SPLINE
SPL {X  -156.487, Y  +349.204, Z    +0.000, E1   +21.338, E3 +377036.669}
SPL {X  -159.136, Y  +365.992, Z    +0.000, E1   +12.463, E3 +377047.428}
SPL {X  -159.799, Y  +374.694, Z    +0.000, E1    +7.504, E3 +377050.531}
SPL {X  -159.976, Y  +380.404, Z    +0.000, E1    +3.959, E3 +377052.064}
SPL {X  -159.990, Y  +384.773, Z    +0.000, E1    +1.003, E3 +377052.959}
SPL {X  -159.990, Y  +387.968, Z    +0.000, E1    -1.448, E3 +377053.527}
SPL {X  -159.990, Y  +391.397, Z    +0.000, E1    -4.422, E3 +377054.151}
SPL {X  -159.990, Y  +395.864, Z    +0.000, E1    -8.712, E3 +377055.240}
SPL {X  -159.990, Y  +401.273, Z    +0.000, E1   -14.176, E3 +377056.967}
SPL {X  -159.990, Y  +409.369, Z    +0.000, E1   -21.807, E3 +377060.759}
SPL {X  -159.990, Y  +436.107, Z    +0.000, E1   -36.921, E3 +377083.684}
SPL {X  -159.990, Y  +469.969, Z    +0.000, E1   -41.961, E3 +377138.388}
SPL {X  -159.990, Y  +477.498, Z    +0.000, E1   -41.916, E3 +377156.272}
SPL {X  -159.990, Y  +483.140, Z    +0.000, E1   -41.902, E3 +377169.628}
SPL {X  -159.990, Y  +488.618, Z    +0.000, E1   -41.913, E3 +377182.559}
SPL {X  -159.990, Y  +494.299, Z    +0.000, E1   -41.910, E3 +377195.994}
SPL {X  -159.990, Y  +499.538, Z    +0.000, E1   -41.904, E3 +377208.388}
SPL {X  -159.990, Y  +505.259, Z    +0.000, E1   -41.922, E3 +377221.887}
SPL {X  -159.990, Y  +511.862, Z    +0.000, E1   -41.927, E3 +377237.498}
SPL {X  -159.990, Y  +519.146, Z    +0.000, E1   -41.942, E3 +377254.691}
SPL {X  -159.990, Y  +526.974, Z    +0.000, E1   -41.950, E3 +377273.191}
SPL {X  -159.990, Y  +533.758, Z    +0.000, E1   -41.910, E3 +377289.294}
SPL {X  -159.990, Y  +539.474, Z    +0.000, E1   -41.912, E3 +377302.821}
SPL {X  -159.990, Y  +544.879, Z    +0.000, E1   -41.899, E3 +377315.633}
SPL {X  -159.990, Y  +550.802, Z    +0.000, E1   -41.920, E3 +377329.614}
SPL {X  -159.990, Y  +556.952, Z    +0.000, E1   -41.911, E3 +377344.153}
SPL {X  -159.990, Y  +562.629, Z    +0.000, E1   -41.910, E3 +377357.571}
SPL {X  -159.990, Y  +567.682, Z    +0.000, E1   -41.901, E3 +377369.530}
SPL {X  -159.990, Y  +572.912, Z    +0.000, E1   -41.914, E3 +377381.877}
SPL {X  -159.990, Y  +578.863, Z    +0.000, E1   -41.918, E3 +377395.941}
SPL {X  -159.990, Y  +584.320, Z    +0.000, E1   -41.901, E3 +377408.888}
SPL {X  -159.990, Y  +589.217, Z    +0.000, E1   -41.901, E3 +377420.461}
SPL {X  -159.990, Y  +594.252, Z    +0.000, E1   -41.903, E3 +377432.376}
SPL {X  -159.990, Y  +600.237, Z    +0.000, E1   -41.928, E3 +377446.493}
SPL {X  -159.990, Y  +607.478, Z    +0.000, E1   -41.933, E3 +377463.602}
SPL {X  -159.990, Y  +614.570, Z    +0.000, E1   -41.926, E3 +377480.383}
SPL {X  -159.990, Y  +621.417, Z    +0.000, E1   -41.931, E3 +377496.576}
SPL {X  -159.990, Y  +627.900, Z    +0.000, E1   -41.914, E3 +377511.916}
SPL {X  -159.990, Y  +634.411, Z    +0.000, E1   -41.931, E3 +377527.285}
SPL {X  -159.990, Y  +641.479, Z    +0.000, E1   -41.931, E3 +377544.002}
SPL {X  -159.990, Y  +647.782, Z    +0.000, E1   -41.914, E3 +377558.923}
SPL {X  -159.990, Y  +653.094, Z    +0.000, E1   -41.905, E3 +377571.502}
SPL {X  -159.990, Y  +657.893, Z    +0.000, E1   -41.899, E3 +377582.867}
SPL {X  -159.990, Y  +662.516, Z    +0.000, E1   -41.899, E3 +377593.799}
SPL {X  -159.990, Y  +668.411, Z    +0.000, E1   -41.929, E3 +377607.692}
SPL {X  -159.968, Y  +674.139, Z    +0.000, E1   -41.898, E3 +377621.296}
SPL {X  -159.817, Y  +678.937, Z    +0.000, E1   -41.879, E3 +377632.793}
SPL {X  -159.484, Y  +684.213, Z    +0.000, E1   -41.818, E3 +377645.629}
SPL {X  -159.007, Y  +689.209, Z    +0.000, E1   -41.732, E3 +377657.934}
SPL {X  -158.327, Y  +694.511, Z    +0.000, E1   -41.622, E3 +377671.184}
SPL {X  -157.480, Y  +699.729, Z    +0.000, E1   -41.453, E3 +377684.447}
SPL {X  -156.604, Y  +704.242, Z    +0.000, E1   -41.288, E3 +377696.056}
SPL {X  -155.514, Y  +709.078, Z    +0.000, E1   -41.107, E3 +377708.610}
SPL {X  -154.232, Y  +714.035, Z    +0.000, E1   -40.861, E3 +377721.669}
SPL {X  -153.147, Y  +717.790, Z    +0.000, E1   -40.640, E3 +377731.687}
SPL {X  -151.881, Y  +721.788, Z    +0.000, E1   -40.435, E3 +377742.374}
SPL {X  -148.572, Y  +730.857, Z    +0.000, E1   -36.304, E3 +377798.582}
ENDSPLINE

SPLINE
SPL {X  -156.377, Y  +705.307, Z    +0.000, E1   -21.740, E3 +377852.831}
SPL {X  -159.301, Y  +686.331, Z    +0.000, E1   -11.648, E3 +377865.476}
SPL {X  -159.936, Y  +675.651, Z    +0.000, E1    -5.377, E3 +377869.192}
SPL {X  -159.990, Y  +670.142, Z    +0.000, E1    -1.740, E3 +377870.491}
SPL {X  -159.990, Y  +666.629, Z    +0.000, E1    +0.827, E3 +377871.140}
SPL {X  -159.990, Y  +662.407, Z    +0.000, E1    +4.406, E3 +377871.991}
SPL {X  -159.990, Y  +655.884, Z    +0.000, E1   +10.601, E3 +377873.856}
SPL {X  -159.990, Y  +646.242, Z    +0.000, E1   +19.956, E3 +377877.775}
SPL {X  -159.990, Y  +624.365, Z    +0.000, E1   +33.860, E3 +377895.677}
SPL {X  -159.990, Y  +615.596, Z    +0.000, E1   +36.980, E3 +377905.336}
SPL {X  -159.990, Y  +586.905, Z    +0.000, E1   +41.264, E3 +377952.362}
SPL {X  -159.990, Y  +581.111, Z    +0.000, E1   +41.245, E3 +377966.416}
SPL {X  -159.990, Y  +576.269, Z    +0.000, E1   +41.239, E3 +377978.143}
SPL {X  -159.990, Y  +571.714, Z    +0.000, E1   +41.240, E3 +377989.171}
SPL {X  -159.990, Y  +567.050, Z    +0.000, E1   +41.238, E3 +378000.458}
SPL {X  -159.990, Y  +561.959, Z    +0.000, E1   +41.251, E3 +378012.757}
SPL {X  -159.990, Y  +557.719, Z    +0.000, E1   +41.226, E3 +378023.059}
SPL {X  -159.990, Y  +554.148, Z    +0.000, E1   +41.237, E3 +378031.674}
SPL {X  -159.990, Y  +548.812, Z    +0.000, E1   +41.263, E3 +378044.549}
SPL {X  -159.990, Y  +542.097, Z    +0.000, E1   +41.274, E3 +378060.801}
SPL {X  -159.990, Y  +535.325, Z    +0.000, E1   +41.260, E3 +378077.202}
SPL {X  -159.990, Y  +529.136, Z    +0.000, E1   +41.262, E3 +378092.170}
SPL {X  -159.990, Y  +524.776, Z    +0.000, E1   +41.225, E3 +378102.783}
SPL {X  -159.990, Y  +521.454, Z    +0.000, E1   +41.236, E3 +378110.805}
SPL {X  -159.990, Y  +515.605, Z    +0.000, E1   +41.288, E3 +378124.844}
SPL {X  -159.990, Y  +509.898, Z    +0.000, E1   +41.246, E3 +378138.706}
SPL {X  -159.990, Y  +505.215, Z    +0.000, E1   +41.261, E3 +378150.022}
SPL {X  -159.990, Y  +500.102, Z    +0.000, E1   +41.251, E3 +378162.405}
SPL {X  -159.990, Y  +495.023, Z    +0.000, E1   +41.263, E3 +378174.654}
SPL {X  -159.990, Y  +479.011, Z    +0.000, E1   +45.740, E3 +378184.036}
SPL {X  -159.990, Y  +471.379, Z    +0.000, E1   +46.435, E3 +378195.651}
SPL {X  -159.990, Y  +466.895, Z    +0.000, E1   +45.533, E3 +378210.056}
SPL {X  -159.990, Y  +462.409, Z    +0.000, E1   +44.664, E3 +378224.831}
SPL {X  -159.990, Y  +458.229, Z    +0.000, E1   +43.579, E3 +378240.313}
SPL {X  -159.990, Y  +453.434, Z    +0.000, E1   +43.227, E3 +378253.087}
SPL {X  -159.990, Y  +448.702, Z    +0.000, E1   +43.218, E3 +378263.809}
SPL {X  -159.990, Y  +442.224, Z    +0.000, E1   +43.270, E3 +378278.359}
SPL {X  -159.990, Y  +435.724, Z    +0.000, E1   +43.218, E3 +378293.117}
SPL {X  -159.990, Y  +430.527, Z    +0.000, E1   +43.236, E3 +378304.807}
SPL {X  -159.990, Y  +424.433, Z    +0.000, E1   +43.237, E3 +378318.556}
SPL {X  -159.990, Y  +419.466, Z    +0.000, E1   +43.217, E3 +378329.795}
SPL {X  -159.990, Y  +414.585, Z    +0.000, E1   +43.233, E3 +378340.787}
SPL {X  -159.990, Y  +409.927, Z    +0.000, E1   +43.217, E3 +378351.319}
SPL {X  -159.990, Y  +405.428, Z    +0.000, E1   +43.230, E3 +378361.477}
SPL {X  -159.990, Y  +398.518, Z    +0.000, E1   +43.261, E3 +378377.032}
SPL {X  -159.990, Y  +392.163, Z    +0.000, E1   +43.223, E3 +378391.432}
SPL {X  -159.990, Y  +387.342, Z    +0.000, E1   +43.224, E3 +378402.309}
SPL {X  -159.990, Y  +382.548, Z    +0.000, E1   +43.224, E3 +378413.132}
SPL {X  -159.922, Y  +377.835, Z    +0.000, E1   +43.211, E3 +378423.849}
SPL {X  -159.608, Y  +371.448, Z    +0.000, E1   +43.200, E3 +378438.525}
SPL {X  -158.905, Y  +363.898, Z    +0.000, E1   +43.073, E3 +378456.293}
SPL {X  -158.182, Y  +358.518, Z    +0.000, E1   +42.902, E3 +378469.237}
SPL {X  -157.507, Y  +354.423, Z    +0.000, E1   +42.786, E3 +378479.182}
SPL {X  -156.676, Y  +350.104, Z    +0.000, E1   +42.637, E3 +378489.787}
SPL {X  -155.489, Y  +344.819, Z    +0.000, E1   +42.446, E3 +378502.911}
SPL {X  -153.911, Y  +338.816, Z    +0.000, E1   +42.155, E3 +378518.087}
SPL {X  -152.412, Y  +333.846, Z    +0.000, E1   +41.856, E3 +378530.857}
SPL {X  -151.009, Y  +329.651, Z    +0.000, E1   +41.581, E3 +378541.757}
SPL {X  -148.356, Y  +322.607, Z    +0.000, E1   +36.121, E3 +378602.233}
ENDSPLINE

SPLINE
SPL {X  -156.487, Y  +349.204, Z    +0.000, E1   +21.338, E3 +378657.359}
SPL {X  -159.136, Y  +365.992, Z    +0.000, E1   +12.463, E3 +378668.117}
SPL {X  -159.799, Y  +374.694, Z    +0.000, E1    +7.504, E3 +378671.221}
SPL {X  -159.976, Y  +380.404, Z    +0.000, E1    +3.959, E3 +378672.754}
SPL {X  -159.990, Y  +384.773, Z    +0.000, E1    +1.003, E3 +378673.648}
SPL {X  -159.990, Y  +387.968, Z    +0.000, E1    -1.448, E3 +378674.217}
SPL {X  -159.990, Y  +391.397, Z    +0.000, E1    -4.422, E3 +378674.841}
SPL {X  -159.990, Y  +395.864, Z    +0.000, E1    -8.712, E3 +378675.929}
SPL {X  -159.990, Y  +401.273, Z    +0.000, E1   -14.176, E3 +378677.657}
SPL {X  -159.990, Y  +409.369, Z    +0.000, E1   -21.807, E3 +378681.448}
SPL {X  -159.990, Y  +436.107, Z    +0.000, E1   -36.921, E3 +378704.374}
SPL {X  -159.990, Y  +469.969, Z    +0.000, E1   -41.961, E3 +378759.078}
SPL {X  -159.990, Y  +477.498, Z    +0.000, E1   -41.916, E3 +378776.962}
SPL {X  -159.990, Y  +483.140, Z    +0.000, E1   -41.902, E3 +378790.317}
SPL {X  -159.990, Y  +488.618, Z    +0.000, E1   -41.913, E3 +378803.249}
SPL {X  -159.990, Y  +494.299, Z    +0.000, E1   -41.910, E3 +378816.683}
SPL {X  -159.990, Y  +499.538, Z    +0.000, E1   -41.904, E3 +378829.078}
SPL {X  -159.990, Y  +504.097, Z    +0.000, E1   -41.897, E3 +378839.866}
SPL {X  -159.990, Y  +509.413, Z    +0.000, E1   -41.921, E3 +378852.401}
SPL {X  -159.990, Y  +516.193, Z    +0.000, E1   -41.932, E3 +378868.417}
SPL {X  -159.990, Y  +523.027, Z    +0.000, E1   -41.926, E3 +378884.579}
SPL {X  -159.990, Y  +528.611, Z    +0.000, E1   -41.900, E3 +378897.834}
SPL {X  -159.990, Y  +533.758, Z    +0.000, E1   -41.910, E3 +378909.983}
SPL {X  -159.990, Y  +539.474, Z    +0.000, E1   -41.912, E3 +378923.511}
SPL {X  -159.990, Y  +544.879, Z    +0.000, E1   -41.899, E3 +378936.322}
SPL {X  -159.990, Y  +550.802, Z    +0.000, E1   -41.920, E3 +378950.304}
SPL {X  -159.990, Y  +556.952, Z    +0.000, E1   -41.911, E3 +378964.843}
SPL {X  -159.990, Y  +562.629, Z    +0.000, E1   -41.910, E3 +378978.261}
SPL {X  -159.990, Y  +567.682, Z    +0.000, E1   -41.901, E3 +378990.220}
SPL {X  -159.990, Y  +574.350, Z    +0.000, E1   -41.955, E3 +379005.905}
SPL {X  -159.990, Y  +580.118, Z    +0.000, E1   -41.891, E3 +379019.642}
SPL {X  -159.990, Y  +584.320, Z    +0.000, E1   -41.901, E3 +379029.578}
SPL {X  -159.990, Y  +589.217, Z    +0.000, E1   -41.901, E3 +379041.151}
SPL {X  -159.990, Y  +594.252, Z    +0.000, E1   -41.903, E3 +379053.065}
SPL {X  -159.990, Y  +600.237, Z    +0.000, E1   -41.928, E3 +379067.183}
SPL {X  -159.990, Y  +605.518, Z    +0.000, E1   -41.890, E3 +379079.721}
SPL {X  -159.990, Y  +610.545, Z    +0.000, E1   -41.917, E3 +379091.569}
SPL {X  -159.990, Y  +615.720, Z    +0.000, E1   -41.899, E3 +379103.829}
SPL {X  -159.990, Y  +620.005, Z    +0.000, E1   -41.900, E3 +379113.962}
SPL {X  -159.990, Y  +624.919, Z    +0.000, E1   -41.912, E3 +379125.569}
SPL {X  -159.990, Y  +629.282, Z    +0.000, E1   -41.888, E3 +379135.910}
SPL {X  -159.990, Y  +632.270, Z    +0.000, E1   -41.887, E3 +379142.982}
SPL {X  -159.990, Y  +637.009, Z    +0.000, E1   -41.925, E3 +379154.124}
SPL {X  -159.990, Y  +642.624, Z    +0.000, E1   -41.901, E3 +379167.445}
SPL {X  -159.990, Y  +647.782, Z    +0.000, E1   -41.914, E3 +379179.613}
SPL {X  -159.990, Y  +653.094, Z    +0.000, E1   -41.905, E3 +379192.191}
SPL {X  -159.990, Y  +657.893, Z    +0.000, E1   -41.899, E3 +379203.557}
SPL {X  -159.990, Y  +662.516, Z    +0.000, E1   -41.899, E3 +379214.488}
SPL {X  -159.990, Y  +666.974, Z    +0.000, E1   -41.897, E3 +379225.033}
SPL {X  -159.984, Y  +672.859, Z    +0.000, E1   -41.934, E3 +379238.894}
SPL {X  -159.817, Y  +678.937, Z    +0.000, E1   -41.879, E3 +379253.482}
SPL {X  -159.484, Y  +684.213, Z    +0.000, E1   -41.818, E3 +379266.318}
SPL {X  -159.007, Y  +689.209, Z    +0.000, E1   -41.732, E3 +379278.623}
SPL {X  -158.485, Y  +693.390, Z    +0.000, E1   -41.627, E3 +379289.076}
SPL {X  -157.663, Y  +698.690, Z    +0.000, E1   -41.523, E3 +379302.438}
SPL {X  -156.604, Y  +704.242, Z    +0.000, E1   -41.288, E3 +379316.746}
SPL {X  -155.831, Y  +707.744, Z    +0.000, E1   -41.132, E3 +379325.866}
SPL {X  -155.167, Y  +710.488, Z    +0.000, E1   -41.008, E3 +379333.044}
SPL {X  -154.232, Y  +714.035, Z    +0.000, E1   -40.861, E3 +379342.358}
SPL {X  -153.147, Y  +717.790, Z    +0.000, E1   -40.640, E3 +379352.377}
SPL {X  -151.881, Y  +721.788, Z    +0.000, E1   -40.435, E3 +379363.063}
SPL {X  -148.572, Y  +730.857, Z    +0.000, E1   -36.304, E3 +379419.272}
ENDSPLINE

SPLINE
SPL {X  -156.377, Y  +705.307, Z    +0.000, E1   -21.740, E3 +379473.521}
SPL {X  -158.965, Y  +689.585, Z    +0.000, E1   -13.405, E3 +379484.678}
SPL {X  -159.884, Y  +677.314, Z    +0.000, E1    -6.475, E3 +379489.391}
SPL {X  -159.990, Y  +670.142, Z    +0.000, E1    -1.740, E3 +379491.180}
SPL {X  -159.990, Y  +666.629, Z    +0.000, E1    +0.827, E3 +379491.830}
SPL {X  -159.990, Y  +662.407, Z    +0.000, E1    +4.406, E3 +379492.680}
SPL {X  -159.990, Y  +655.884, Z    +0.000, E1   +10.601, E3 +379494.546}
SPL {X  -159.990, Y  +643.833, Z    +0.000, E1   +21.883, E3 +379500.175}
SPL {X  -159.990, Y  +617.235, Z    +0.000, E1   +36.481, E3 +379524.075}
SPL {X  -159.990, Y  +586.905, Z    +0.000, E1   +41.264, E3 +379573.051}
SPL {X  -159.990, Y  +581.111, Z    +0.000, E1   +41.245, E3 +379587.105}
SPL {X  -159.990, Y  +576.269, Z    +0.000, E1   +41.239, E3 +379598.833}
SPL {X  -159.990, Y  +571.714, Z    +0.000, E1   +41.240, E3 +379609.861}
SPL {X  -159.990, Y  +567.050, Z    +0.000, E1   +41.238, E3 +379621.148}
SPL {X  -159.990, Y  +561.959, Z    +0.000, E1   +41.251, E3 +379633.446}
SPL {X  -159.990, Y  +557.719, Z    +0.000, E1   +41.226, E3 +379643.749}
SPL {X  -159.990, Y  +554.148, Z    +0.000, E1   +41.237, E3 +379652.364}
SPL {X  -159.990, Y  +548.812, Z    +0.000, E1   +41.263, E3 +379665.238}
SPL {X  -159.990, Y  +543.804, Z    +0.000, E1   +41.237, E3 +379677.403}
SPL {X  -159.990, Y  +538.952, Z    +0.000, E1   +41.247, E3 +379689.150}
SPL {X  -159.990, Y  +534.225, Z    +0.000, E1   +41.236, E3 +379700.584}
SPL {X  -159.990, Y  +529.136, Z    +0.000, E1   +41.262, E3 +379712.859}
SPL {X  -159.990, Y  +522.690, Z    +0.000, E1   +41.265, E3 +379728.459}
SPL {X  -159.990, Y  +516.698, Z    +0.000, E1   +41.259, E3 +379742.933}
SPL {X  -159.990, Y  +510.896, Z    +0.000, E1   +41.267, E3 +379756.951}
SPL {X  -159.990, Y  +505.215, Z    +0.000, E1   +41.261, E3 +379770.711}
SPL {X  -159.990, Y  +500.102, Z    +0.000, E1   +41.251, E3 +379783.094}
SPL {X  -159.990, Y  +495.023, Z    +0.000, E1   +41.263, E3 +379795.343}
SPL {X  -159.990, Y  +479.011, Z    +0.000, E1   +45.740, E3 +379804.725}
SPL {X  -159.990, Y  +471.379, Z    +0.000, E1   +46.435, E3 +379816.341}
SPL {X  -159.990, Y  +466.895, Z    +0.000, E1   +45.533, E3 +379830.745}
SPL {X  -159.990, Y  +462.409, Z    +0.000, E1   +44.664, E3 +379845.520}
SPL {X  -159.990, Y  +458.229, Z    +0.000, E1   +43.579, E3 +379861.003}
SPL {X  -159.990, Y  +453.434, Z    +0.000, E1   +43.227, E3 +379873.777}
SPL {X  -159.990, Y  +448.702, Z    +0.000, E1   +43.218, E3 +379884.499}
SPL {X  -159.990, Y  +444.476, Z    +0.000, E1   +43.219, E3 +379894.037}
SPL {X  -159.990, Y  +440.246, Z    +0.000, E1   +43.217, E3 +379903.595}
SPL {X  -159.990, Y  +434.411, Z    +0.000, E1   +43.246, E3 +379916.725}
SPL {X  -159.990, Y  +429.216, Z    +0.000, E1   +43.210, E3 +379928.498}
SPL {X  -159.990, Y  +424.433, Z    +0.000, E1   +43.237, E3 +379939.245}
SPL {X  -159.990, Y  +419.466, Z    +0.000, E1   +43.217, E3 +379950.485}
SPL {X  -159.990, Y  +414.585, Z    +0.000, E1   +43.233, E3 +379961.477}
SPL {X  -159.990, Y  +409.927, Z    +0.000, E1   +43.217, E3 +379972.009}
SPL {X  -159.990, Y  +405.428, Z    +0.000, E1   +43.230, E3 +379982.167}
SPL {X  -159.990, Y  +398.518, Z    +0.000, E1   +43.261, E3 +379997.721}
SPL {X  -159.990, Y  +392.163, Z    +0.000, E1   +43.223, E3 +380012.121}
SPL {X  -159.990, Y  +387.342, Z    +0.000, E1   +43.224, E3 +380022.999}
SPL {X  -159.990, Y  +382.548, Z    +0.000, E1   +43.224, E3 +380033.821}
SPL {X  -159.922, Y  +377.835, Z    +0.000, E1   +43.211, E3 +380044.538}
SPL {X  -159.712, Y  +373.072, Z    +0.000, E1   +43.177, E3 +380055.504}
SPL {X  -159.289, Y  +367.537, Z    +0.000, E1   +43.118, E3 +380068.416}
SPL {X  -158.730, Y  +362.464, Z    +0.000, E1   +43.003, E3 +380080.448}
SPL {X  -158.182, Y  +358.518, Z    +0.000, E1   +42.902, E3 +380089.926}
SPL {X  -157.507, Y  +354.423, Z    +0.000, E1   +42.786, E3 +380099.872}
SPL {X  -156.676, Y  +350.104, Z    +0.000, E1   +42.637, E3 +380110.477}
SPL {X  -155.807, Y  +346.154, Z    +0.000, E1   +42.470, E3 +380120.304}
SPL {X  -154.777, Y  +341.993, Z    +0.000, E1   +42.302, E3 +380130.729}
SPL {X  -153.585, Y  +337.686, Z    +0.000, E1   +42.062, E3 +380141.705}
SPL {X  -152.412, Y  +333.846, Z    +0.000, E1   +41.856, E3 +380151.547}
SPL {X  -151.009, Y  +329.651, Z    +0.000, E1   +41.581, E3 +380162.447}
SPL {X  -148.356, Y  +322.607, Z    +0.000, E1   +36.121, E3 +380222.923}
ENDSPLINE

SPLINE
SPL {X  -156.487, Y  +349.204, Z    +0.000, E1   +21.338, E3 +380278.048}
SPL {X  -159.136, Y  +365.992, Z    +0.000, E1   +12.463, E3 +380288.807}
SPL {X  -159.799, Y  +374.694, Z    +0.000, E1    +7.504, E3 +380291.911}
SPL {X  -159.976, Y  +380.404, Z    +0.000, E1    +3.959, E3 +380293.444}
SPL {X  -159.990, Y  +384.773, Z    +0.000, E1    +1.003, E3 +380294.338}
SPL {X  -159.990, Y  +387.968, Z    +0.000, E1    -1.448, E3 +380294.906}
SPL {X  -159.990, Y  +391.397, Z    +0.000, E1    -4.422, E3 +380295.530}
SPL {X  -159.990, Y  +395.864, Z    +0.000, E1    -8.712, E3 +380296.619}
SPL {X  -159.990, Y  +401.273, Z    +0.000, E1   -14.176, E3 +380298.346}
SPL {X  -159.990, Y  +411.788, Z    +0.000, E1   -23.693, E3 +380303.889}
SPL {X  -159.990, Y  +438.158, Z    +0.000, E1   -37.630, E3 +380327.167}
SPL {X  -159.990, Y  +468.567, Z    +0.000, E1   -41.922, E3 +380376.510}
SPL {X  -159.990, Y  +474.616, Z    +0.000, E1   -41.909, E3 +380390.840}
SPL {X  -159.990, Y  +481.610, Z    +0.000, E1   -41.947, E3 +380407.326}
SPL {X  -159.990, Y  +488.618, Z    +0.000, E1   -41.913, E3 +380423.939}
SPL {X  -159.990, Y  +494.299, Z    +0.000, E1   -41.910, E3 +380437.373}
SPL {X  -159.990, Y  +499.538, Z    +0.000, E1   -41.904, E3 +380449.767}
SPL {X  -159.990, Y  +505.259, Z    +0.000, E1   -41.922, E3 +380463.267}
SPL {X  -159.990, Y  +511.862, Z    +0.000, E1   -41.927, E3 +380478.877}
SPL {X  -159.990, Y  +517.450, Z    +0.000, E1   -41.901, E3 +380492.124}
SPL {X  -159.990, Y  +523.027, Z    +0.000, E1   -41.926, E3 +380505.269}
SPL {X  -159.990, Y  +528.611, Z    +0.000, E1   -41.900, E3 +380518.524}
SPL {X  -159.990, Y  +533.758, Z    +0.000, E1   -41.910, E3 +380530.673}
SPL {X  -159.990, Y  +539.474, Z    +0.000, E1   -41.912, E3 +380544.200}
SPL {X  -159.990, Y  +544.879, Z    +0.000, E1   -41.899, E3 +380557.012}
SPL {X  -159.990, Y  +550.802, Z    +0.000, E1   -41.920, E3 +380570.993}
SPL {X  -159.990, Y  +556.952, Z    +0.000, E1   -41.911, E3 +380585.532}
SPL {X  -159.990, Y  +562.629, Z    +0.000, E1   -41.910, E3 +380598.950}
SPL {X  -159.990, Y  +567.682, Z    +0.000, E1   -41.901, E3 +380610.909}
SPL {X  -159.990, Y  +572.912, Z    +0.000, E1   -41.914, E3 +380623.257}
SPL {X  -159.990, Y  +578.863, Z    +0.000, E1   -41.918, E3 +380637.321}
SPL {X  -159.990, Y  +584.320, Z    +0.000, E1   -41.901, E3 +380650.267}
SPL {X  -159.990, Y  +589.217, Z    +0.000, E1   -41.901, E3 +380661.840}
SPL {X  -159.990, Y  +594.252, Z    +0.000, E1   -41.903, E3 +380673.755}
SPL {X  -159.990, Y  +598.793, Z    +0.000, E1   -41.896, E3 +380684.509}
SPL {X  -159.990, Y  +604.215, Z    +0.000, E1   -41.919, E3 +380697.289}
SPL {X  -159.990, Y  +609.216, Z    +0.000, E1   -41.890, E3 +380709.157}
SPL {X  -159.990, Y  +614.570, Z    +0.000, E1   -41.926, E3 +380721.762}
SPL {X  -159.990, Y  +620.005, Z    +0.000, E1   -41.900, E3 +380734.652}
SPL {X  -159.990, Y  +624.919, Z    +0.000, E1   -41.912, E3 +380746.259}
SPL {X  -159.990, Y  +630.816, Z    +0.000, E1   -41.915, E3 +380760.188}
SPL {X  -159.990, Y  +637.009, Z    +0.000, E1   -41.925, E3 +380774.814}
SPL {X  -159.990, Y  +642.624, Z    +0.000, E1   -41.901, E3 +380788.134}
SPL {X  -159.990, Y  +647.782, Z    +0.000, E1   -41.914, E3 +380800.303}
SPL {X  -159.990, Y  +653.094, Z    +0.000, E1   -41.905, E3 +380812.881}
SPL {X  -159.990, Y  +657.893, Z    +0.000, E1   -41.899, E3 +380824.247}
SPL {X  -159.990, Y  +662.516, Z    +0.000, E1   -41.899, E3 +380835.178}
SPL {X  -159.990, Y  +666.974, Z    +0.000, E1   -41.897, E3 +380845.722}
SPL {X  -159.984, Y  +672.859, Z    +0.000, E1   -41.934, E3 +380859.584}
SPL {X  -159.817, Y  +678.937, Z    +0.000, E1   -41.879, E3 +380874.172}
SPL {X  -159.484, Y  +684.213, Z    +0.000, E1   -41.818, E3 +380887.008}
SPL {X  -159.007, Y  +689.209, Z    +0.000, E1   -41.732, E3 +380899.313}
SPL {X  -158.327, Y  +694.511, Z    +0.000, E1   -41.622, E3 +380912.564}
SPL {X  -157.480, Y  +699.729, Z    +0.000, E1   -41.453, E3 +380925.827}
SPL {X  -156.604, Y  +704.242, Z    +0.000, E1   -41.288, E3 +380937.435}
SPL {X  -155.514, Y  +709.078, Z    +0.000, E1   -41.107, E3 +380949.989}
SPL {X  -154.232, Y  +714.035, Z    +0.000, E1   -40.861, E3 +380963.048}
SPL {X  -153.147, Y  +717.790, Z    +0.000, E1   -40.640, E3 +380973.066}
SPL {X  -151.881, Y  +721.788, Z    +0.000, E1   -40.435, E3 +380983.753}
SPL {X  -148.572, Y  +730.857, Z    +0.000, E1   -36.304, E3 +381039.962}
ENDSPLINE

SPLINE
SPL {X  -156.377, Y  +705.307, Z    +0.000, E1   -21.740, E3 +381094.210}
SPL {X  -158.965, Y  +689.585, Z    +0.000, E1   -13.405, E3 +381105.368}
SPL {X  -159.884, Y  +677.314, Z    +0.000, E1    -6.475, E3 +381110.081}
SPL {X  -159.990, Y  +670.142, Z    +0.000, E1    -1.740, E3 +381111.870}
SPL {X  -159.990, Y  +666.629, Z    +0.000, E1    +0.827, E3 +381112.520}
SPL {X  -159.990, Y  +662.407, Z    +0.000, E1    +4.406, E3 +381113.370}
SPL {X  -159.990, Y  +655.884, Z    +0.000, E1   +10.601, E3 +381115.235}
SPL {X  -159.990, Y  +643.833, Z    +0.000, E1   +21.883, E3 +381120.864}
SPL {X  -159.990, Y  +617.235, Z    +0.000, E1   +36.481, E3 +381144.765}
SPL {X  -159.990, Y  +586.905, Z    +0.000, E1   +41.264, E3 +381193.741}
SPL {X  -159.990, Y  +581.111, Z    +0.000, E1   +41.245, E3 +381207.795}
SPL {X  -159.990, Y  +576.269, Z    +0.000, E1   +41.239, E3 +381219.523}
SPL {X  -159.990, Y  +571.714, Z    +0.000, E1   +41.240, E3 +381230.551}
SPL {X  -159.990, Y  +567.050, Z    +0.000, E1   +41.238, E3 +381241.837}
SPL {X  -159.990, Y  +561.959, Z    +0.000, E1   +41.251, E3 +381254.136}
SPL {X  -159.990, Y  +557.719, Z    +0.000, E1   +41.226, E3 +381264.438}
SPL {X  -159.990, Y  +554.148, Z    +0.000, E1   +41.237, E3 +381273.053}
SPL {X  -159.990, Y  +548.812, Z    +0.000, E1   +41.263, E3 +381285.928}
SPL {X  -159.990, Y  +543.804, Z    +0.000, E1   +41.237, E3 +381298.093}
SPL {X  -159.990, Y  +538.952, Z    +0.000, E1   +41.247, E3 +381309.840}
SPL {X  -159.990, Y  +534.225, Z    +0.000, E1   +41.236, E3 +381321.273}
SPL {X  -159.990, Y  +529.136, Z    +0.000, E1   +41.262, E3 +381333.549}
SPL {X  -159.990, Y  +522.690, Z    +0.000, E1   +41.265, E3 +381349.149}
SPL {X  -159.990, Y  +516.698, Z    +0.000, E1   +41.259, E3 +381363.623}
SPL {X  -159.990, Y  +510.896, Z    +0.000, E1   +41.267, E3 +381377.641}
SPL {X  -159.990, Y  +506.621, Z    +0.000, E1   +41.235, E3 +381388.043}
SPL {X  -159.990, Y  +501.314, Z    +0.000, E1   +41.284, E3 +381400.802}
SPL {X  -159.990, Y  +495.023, Z    +0.000, E1   +41.263, E3 +381416.033}
SPL {X  -159.990, Y  +479.011, Z    +0.000, E1   +45.740, E3 +381425.415}
SPL {X  -159.990, Y  +471.379, Z    +0.000, E1   +46.435, E3 +381437.030}
SPL {X  -159.990, Y  +466.895, Z    +0.000, E1   +45.533, E3 +381451.435}
SPL {X  -159.990, Y  +462.409, Z    +0.000, E1   +44.664, E3 +381466.210}
SPL {X  -159.990, Y  +458.229, Z    +0.000, E1   +43.579, E3 +381481.692}
SPL {X  -159.990, Y  +453.434, Z    +0.000, E1   +43.227, E3 +381494.467}
SPL {X  -159.990, Y  +448.702, Z    +0.000, E1   +43.218, E3 +381505.189}
SPL {X  -159.990, Y  +444.476, Z    +0.000, E1   +43.219, E3 +381514.727}
SPL {X  -159.990, Y  +440.246, Z    +0.000, E1   +43.217, E3 +381524.284}
SPL {X  -159.990, Y  +434.411, Z    +0.000, E1   +43.246, E3 +381537.415}
SPL {X  -159.990, Y  +429.216, Z    +0.000, E1   +43.210, E3 +381549.187}
SPL {X  -159.990, Y  +424.433, Z    +0.000, E1   +43.237, E3 +381559.935}
SPL {X  -159.990, Y  +419.466, Z    +0.000, E1   +43.217, E3 +381571.175}
SPL {X  -159.990, Y  +414.585, Z    +0.000, E1   +43.233, E3 +381582.167}
SPL {X  -159.990, Y  +409.927, Z    +0.000, E1   +43.217, E3 +381592.698}
SPL {X  -159.990, Y  +405.428, Z    +0.000, E1   +43.230, E3 +381602.856}
SPL {X  -159.990, Y  +398.518, Z    +0.000, E1   +43.261, E3 +381618.411}
SPL {X  -159.990, Y  +392.163, Z    +0.000, E1   +43.223, E3 +381632.811}
SPL {X  -159.990, Y  +387.342, Z    +0.000, E1   +43.224, E3 +381643.688}
SPL {X  -159.990, Y  +382.548, Z    +0.000, E1   +43.224, E3 +381654.511}
SPL {X  -159.922, Y  +377.835, Z    +0.000, E1   +43.211, E3 +381665.228}
SPL {X  -159.608, Y  +371.448, Z    +0.000, E1   +43.200, E3 +381679.904}
SPL {X  -158.905, Y  +363.898, Z    +0.000, E1   +43.073, E3 +381697.673}
SPL {X  -158.182, Y  +358.518, Z    +0.000, E1   +42.902, E3 +381710.616}
SPL {X  -157.507, Y  +354.423, Z    +0.000, E1   +42.786, E3 +381720.561}
SPL {X  -156.676, Y  +350.104, Z    +0.000, E1   +42.637, E3 +381731.167}
SPL {X  -155.807, Y  +346.154, Z    +0.000, E1   +42.470, E3 +381740.994}
SPL {X  -154.777, Y  +341.993, Z    +0.000, E1   +42.302, E3 +381751.419}
SPL {X  -153.585, Y  +337.686, Z    +0.000, E1   +42.062, E3 +381762.394}
SPL {X  -152.412, Y  +333.846, Z    +0.000, E1   +41.856, E3 +381772.237}
SPL {X  -151.009, Y  +329.651, Z    +0.000, E1   +41.581, E3 +381783.137}
SPL {X  -148.356, Y  +322.607, Z    +0.000, E1   +36.121, E3 +381843.612}
ENDSPLINE

SPLINE
SPL {X  -156.487, Y  +349.204, Z    +0.000, E1   +21.338, E3 +381898.738}
SPL {X  -159.136, Y  +365.992, Z    +0.000, E1   +12.463, E3 +381909.497}
SPL {X  -159.799, Y  +374.694, Z    +0.000, E1    +7.504, E3 +381912.600}
SPL {X  -159.976, Y  +380.404, Z    +0.000, E1    +3.959, E3 +381914.133}
SPL {X  -159.990, Y  +384.773, Z    +0.000, E1    +1.003, E3 +381915.028}
SPL {X  -159.990, Y  +387.968, Z    +0.000, E1    -1.448, E3 +381915.596}
SPL {X  -159.990, Y  +391.397, Z    +0.000, E1    -4.422, E3 +381916.220}
SPL {X  -159.990, Y  +395.864, Z    +0.000, E1    -8.712, E3 +381917.308}
SPL {X  -159.990, Y  +401.273, Z    +0.000, E1   -14.176, E3 +381919.036}
SPL {X  -159.990, Y  +411.788, Z    +0.000, E1   -23.693, E3 +381924.579}
SPL {X  -159.990, Y  +438.158, Z    +0.000, E1   -37.630, E3 +381947.856}
SPL {X  -159.990, Y  +465.724, Z    +0.000, E1   -41.883, E3 +381990.551}
SPL {X  -159.990, Y  +470.837, Z    +0.000, E1   -41.927, E3 +382002.565}
SPL {X  -159.990, Y  +477.498, Z    +0.000, E1   -41.916, E3 +382018.341}
SPL {X  -159.990, Y  +483.140, Z    +0.000, E1   -41.902, E3 +382031.697}
SPL {X  -159.990, Y  +488.618, Z    +0.000, E1   -41.913, E3 +382044.628}
SPL {X  -159.990, Y  +494.299, Z    +0.000, E1   -41.910, E3 +382058.063}
SPL {X  -159.990, Y  +499.538, Z    +0.000, E1   -41.904, E3 +382070.457}
SPL {X  -159.990, Y  +504.097, Z    +0.000, E1   -41.897, E3 +382081.245}
SPL {X  -159.990, Y  +509.413, Z    +0.000, E1   -41.921, E3 +382093.781}
SPL {X  -159.990, Y  +513.834, Z    +0.000, E1   -41.885, E3 +382104.294}
SPL {X  -159.990, Y  +517.450, Z    +0.000, E1   -41.901, E3 +382112.814}
SPL {X  -159.990, Y  +523.027, Z    +0.000, E1   -41.926, E3 +382125.958}
SPL {X  -159.990, Y  +528.611, Z    +0.000, E1   -41.900, E3 +382139.213}
SPL {X  -159.990, Y  +533.758, Z    +0.000, E1   -41.910, E3 +382151.363}
SPL {X  -159.990, Y  +539.474, Z    +0.000, E1   -41.912, E3 +382164.890}
SPL {X  -159.990, Y  +546.447, Z    +0.000, E1   -41.939, E3 +382181.353}
SPL {X  -159.990, Y  +552.220, Z    +0.000, E1   -41.887, E3 +382195.087}
SPL {X  -159.990, Y  +556.952, Z    +0.000, E1   -41.911, E3 +382206.222}
SPL {X  -159.990, Y  +562.629, Z    +0.000, E1   -41.910, E3 +382219.640}
SPL {X  -159.990, Y  +569.054, Z    +0.000, E1   -41.933, E3 +382234.795}
SPL {X  -159.990, Y  +575.562, Z    +0.000, E1   -41.916, E3 +382250.208}
SPL {X  -159.990, Y  +580.118, Z    +0.000, E1   -41.891, E3 +382261.021}
SPL {X  -159.990, Y  +584.320, Z    +0.000, E1   -41.901, E3 +382270.957}
SPL {X  -159.990, Y  +589.217, Z    +0.000, E1   -41.901, E3 +382282.530}
SPL {X  -159.990, Y  +594.252, Z    +0.000, E1   -41.903, E3 +382294.445}
SPL {X  -159.990, Y  +600.237, Z    +0.000, E1   -41.928, E3 +382308.562}
SPL {X  -159.990, Y  +607.478, Z    +0.000, E1   -41.933, E3 +382325.671}
SPL {X  -159.990, Y  +614.570, Z    +0.000, E1   -41.926, E3 +382342.452}
SPL {X  -159.990, Y  +620.005, Z    +0.000, E1   -41.900, E3 +382355.341}
SPL {X  -159.990, Y  +624.919, Z    +0.000, E1   -41.912, E3 +382366.949}
SPL {X  -159.990, Y  +630.816, Z    +0.000, E1   -41.915, E3 +382380.878}
SPL {X  -159.990, Y  +637.009, Z    +0.000, E1   -41.925, E3 +382395.503}
SPL {X  -159.990, Y  +642.624, Z    +0.000, E1   -41.901, E3 +382408.824}
SPL {X  -159.990, Y  +647.782, Z    +0.000, E1   -41.914, E3 +382420.992}
SPL {X  -159.990, Y  +653.094, Z    +0.000, E1   -41.905, E3 +382433.571}
SPL {X  -159.990, Y  +657.893, Z    +0.000, E1   -41.899, E3 +382444.936}
SPL {X  -159.990, Y  +662.516, Z    +0.000, E1   -41.899, E3 +382455.868}
SPL {X  -159.990, Y  +666.974, Z    +0.000, E1   -41.897, E3 +382466.412}
SPL {X  -159.984, Y  +672.859, Z    +0.000, E1   -41.934, E3 +382480.273}
SPL {X  -159.817, Y  +678.937, Z    +0.000, E1   -41.879, E3 +382494.862}
SPL {X  -159.484, Y  +684.213, Z    +0.000, E1   -41.818, E3 +382507.698}
SPL {X  -159.007, Y  +689.209, Z    +0.000, E1   -41.732, E3 +382520.003}
SPL {X  -158.327, Y  +694.511, Z    +0.000, E1   -41.622, E3 +382533.253}
SPL {X  -157.480, Y  +699.729, Z    +0.000, E1   -41.453, E3 +382546.516}
SPL {X  -156.604, Y  +704.242, Z    +0.000, E1   -41.288, E3 +382558.125}
SPL {X  -155.514, Y  +709.078, Z    +0.000, E1   -41.107, E3 +382570.679}
SPL {X  -154.232, Y  +714.035, Z    +0.000, E1   -40.861, E3 +382583.738}
SPL {X  -153.147, Y  +717.790, Z    +0.000, E1   -40.640, E3 +382593.756}
SPL {X  -151.881, Y  +721.788, Z    +0.000, E1   -40.435, E3 +382604.443}
SPL {X  -148.572, Y  +730.857, Z    +0.000, E1   -36.304, E3 +382660.651}
ENDSPLINE

SPLINE
SPL {X  -154.420, Y  +713.347, Z    +0.000, E1   -25.698, E3 +382706.075}
SPL {X  -156.970, Y  +702.437, Z    +0.000, E1   -20.224, E3 +382717.771}
SPL {X  -158.965, Y  +689.585, Z    +0.000, E1   -13.405, E3 +382726.058}
SPL {X  -159.884, Y  +677.314, Z    +0.000, E1    -6.475, E3 +382730.770}
SPL {X  -159.990, Y  +670.142, Z    +0.000, E1    -1.740, E3 +382732.560}
SPL {X  -159.990, Y  +666.629, Z    +0.000, E1    +0.827, E3 +382733.209}
SPL {X  -159.990, Y  +662.407, Z    +0.000, E1    +4.406, E3 +382734.060}
SPL {X  -159.990, Y  +657.382, Z    +0.000, E1    +9.217, E3 +382735.442}
SPL {X  -159.990, Y  +653.255, Z    +0.000, E1   +13.347, E3 +382736.771}
SPL {X  -159.990, Y  +646.242, Z    +0.000, E1   +19.956, E3 +382739.844}
SPL {X  -159.990, Y  +624.365, Z    +0.000, E1   +33.860, E3 +382757.746}
SPL {X  -159.990, Y  +615.596, Z    +0.000, E1   +36.980, E3 +382767.405}
SPL {X  -159.990, Y  +586.905, Z    +0.000, E1   +41.264, E3 +382814.431}
SPL {X  -159.990, Y  +581.111, Z    +0.000, E1   +41.245, E3 +382828.485}
SPL {X  -159.990, Y  +576.269, Z    +0.000, E1   +41.239, E3 +382840.212}
SPL {X  -159.990, Y  +571.714, Z    +0.000, E1   +41.240, E3 +382851.240}
SPL {X  -159.990, Y  +567.050, Z    +0.000, E1   +41.238, E3 +382862.527}
SPL {X  -159.990, Y  +561.959, Z    +0.000, E1   +41.251, E3 +382874.825}
SPL {X  -159.990, Y  +555.553, Z    +0.000, E1   +41.273, E3 +382890.294}
SPL {X  -159.990, Y  +549.897, Z    +0.000, E1   +41.240, E3 +382904.024}
SPL {X  -159.990, Y  +544.775, Z    +0.000, E1   +41.260, E3 +382916.399}
SPL {X  -159.990, Y  +540.176, Z    +0.000, E1   +41.224, E3 +382927.607}
SPL {X  -159.990, Y  +534.009, Z    +0.000, E1   +41.300, E3 +382942.393}
SPL {X  -159.990, Y  +526.579, Z    +0.000, E1   +41.262, E3 +382960.430}
SPL {X  -159.990, Y  +521.454, Z    +0.000, E1   +41.236, E3 +382972.874}
SPL {X  -159.990, Y  +516.698, Z    +0.000, E1   +41.259, E3 +382984.313}
SPL {X  -159.990, Y  +510.896, Z    +0.000, E1   +41.267, E3 +382998.330}
SPL {X  -159.990, Y  +505.215, Z    +0.000, E1   +41.261, E3 +383012.091}
SPL {X  -159.990, Y  +498.837, Z    +0.000, E1   +41.283, E3 +383027.479}
SPL {X  -159.990, Y  +493.848, Z    +0.000, E1   +41.241, E3 +383039.599}
SPL {X  -159.990, Y  +474.734, Z    +0.000, E1   +46.319, E3 +383051.522}
SPL {X  -159.990, Y  +469.870, Z    +0.000, E1   +46.059, E3 +383062.745}
SPL {X  -159.990, Y  +465.881, Z    +0.000, E1   +45.385, E3 +383075.323}
SPL {X  -159.990, Y  +461.571, Z    +0.000, E1   +44.440, E3 +383089.848}
SPL {X  -159.990, Y  +458.229, Z    +0.000, E1   +43.579, E3 +383102.382}
SPL {X  -159.990, Y  +453.434, Z    +0.000, E1   +43.227, E3 +383115.156}
SPL {X  -159.990, Y  +448.702, Z    +0.000, E1   +43.218, E3 +383125.878}
SPL {X  -159.990, Y  +442.224, Z    +0.000, E1   +43.270, E3 +383140.428}
SPL {X  -159.990, Y  +435.724, Z    +0.000, E1   +43.218, E3 +383155.186}
SPL {X  -159.990, Y  +430.527, Z    +0.000, E1   +43.236, E3 +383166.876}
SPL {X  -159.990, Y  +424.433, Z    +0.000, E1   +43.237, E3 +383180.625}
SPL {X  -159.990, Y  +419.466, Z    +0.000, E1   +43.217, E3 +383191.864}
SPL {X  -159.990, Y  +414.585, Z    +0.000, E1   +43.233, E3 +383202.856}
SPL {X  -159.990, Y  +409.927, Z    +0.000, E1   +43.217, E3 +383213.388}
SPL {X  -159.990, Y  +405.428, Z    +0.000, E1   +43.230, E3 +383223.546}
SPL {X  -159.990, Y  +398.518, Z    +0.000, E1   +43.261, E3 +383239.101}
SPL {X  -159.990, Y  +392.163, Z    +0.000, E1   +43.223, E3 +383253.501}
SPL {X  -159.990, Y  +387.342, Z    +0.000, E1   +43.224, E3 +383264.378}
SPL {X  -159.990, Y  +382.548, Z    +0.000, E1   +43.224, E3 +383275.201}
SPL {X  -159.922, Y  +377.835, Z    +0.000, E1   +43.211, E3 +383285.918}
SPL {X  -159.712, Y  +373.072, Z    +0.000, E1   +43.177, E3 +383296.883}
SPL {X  -159.289, Y  +367.537, Z    +0.000, E1   +43.118, E3 +383309.795}
SPL {X  -158.730, Y  +362.464, Z    +0.000, E1   +43.003, E3 +383321.827}
SPL {X  -158.182, Y  +358.518, Z    +0.000, E1   +42.902, E3 +383331.306}
SPL {X  -157.507, Y  +354.423, Z    +0.000, E1   +42.786, E3 +383341.251}
SPL {X  -156.676, Y  +350.104, Z    +0.000, E1   +42.637, E3 +383351.856}
SPL {X  -155.807, Y  +346.154, Z    +0.000, E1   +42.470, E3 +383361.683}
SPL {X  -154.777, Y  +341.993, Z    +0.000, E1   +42.302, E3 +383372.109}
SPL {X  -153.585, Y  +337.686, Z    +0.000, E1   +42.062, E3 +383383.084}
SPL {X  -152.412, Y  +333.846, Z    +0.000, E1   +41.856, E3 +383392.926}
SPL {X  -151.009, Y  +329.651, Z    +0.000, E1   +41.581, E3 +383403.826}
SPL {X  -148.356, Y  +322.607, Z    +0.000, E1   +36.121, E3 +383464.302}
ENDSPLINE

SPLINE
SPL {X  -156.487, Y  +349.204, Z    +0.000, E1   +21.338, E3 +383519.428}
SPL {X  -159.136, Y  +365.992, Z    +0.000, E1   +12.463, E3 +383530.186}
SPL {X  -159.799, Y  +374.694, Z    +0.000, E1    +7.504, E3 +383533.290}
SPL {X  -159.976, Y  +380.404, Z    +0.000, E1    +3.959, E3 +383534.823}
SPL {X  -159.990, Y  +384.773, Z    +0.000, E1    +1.003, E3 +383535.717}
SPL {X  -159.990, Y  +387.968, Z    +0.000, E1    -1.448, E3 +383536.286}
SPL {X  -159.990, Y  +391.397, Z    +0.000, E1    -4.422, E3 +383536.910}
SPL {X  -159.990, Y  +395.864, Z    +0.000, E1    -8.712, E3 +383537.998}
SPL {X  -159.990, Y  +401.273, Z    +0.000, E1   -14.176, E3 +383539.726}
SPL {X  -159.990, Y  +411.788, Z    +0.000, E1   -23.693, E3 +383545.269}
SPL {X  -159.990, Y  +438.158, Z    +0.000, E1   -37.630, E3 +383568.546}
SPL {X  -159.990, Y  +468.567, Z    +0.000, E1   -41.922, E3 +383617.890}
SPL {X  -159.990, Y  +474.616, Z    +0.000, E1   -41.909, E3 +383632.219}
SPL {X  -159.990, Y  +481.610, Z    +0.000, E1   -41.947, E3 +383648.706}
SPL {X  -159.990, Y  +488.618, Z    +0.000, E1   -41.913, E3 +383665.318}
SPL {X  -159.990, Y  +494.299, Z    +0.000, E1   -41.910, E3 +383678.752}
SPL {X  -159.990, Y  +499.538, Z    +0.000, E1   -41.904, E3 +383691.147}
SPL {X  -159.990, Y  +505.259, Z    +0.000, E1   -41.922, E3 +383704.646}
SPL {X  -159.990, Y  +511.862, Z    +0.000, E1   -41.927, E3 +383720.256}
SPL {X  -159.990, Y  +517.450, Z    +0.000, E1   -41.901, E3 +383733.504}
SPL {X  -159.990, Y  +523.027, Z    +0.000, E1   -41.926, E3 +383746.648}
SPL {X  -159.990, Y  +528.611, Z    +0.000, E1   -41.900, E3 +383759.903}
SPL {X  -159.990, Y  +533.758, Z    +0.000, E1   -41.910, E3 +383772.052}
SPL {X  -159.990, Y  +539.474, Z    +0.000, E1   -41.912, E3 +383785.580}
SPL {X  -159.990, Y  +544.879, Z    +0.000, E1   -41.899, E3 +383798.391}
SPL {X  -159.990, Y  +550.802, Z    +0.000, E1   -41.920, E3 +383812.373}
SPL {X  -159.990, Y  +556.952, Z    +0.000, E1   -41.911, E3 +383826.912}
SPL {X  -159.990, Y  +562.629, Z    +0.000, E1   -41.910, E3 +383840.330}
SPL {X  -159.990, Y  +567.682, Z    +0.000, E1   -41.901, E3 +383852.289}
SPL {X  -159.990, Y  +572.912, Z    +0.000, E1   -41.914, E3 +383864.636}
SPL {X  -159.990, Y  +578.863, Z    +0.000, E1   -41.918, E3 +383878.700}
SPL {X  -159.990, Y  +584.320, Z    +0.000, E1   -41.901, E3 +383891.647}
SPL {X  -159.990, Y  +589.217, Z    +0.000, E1   -41.901, E3 +383903.220}
SPL {X  -159.990, Y  +594.252, Z    +0.000, E1   -41.903, E3 +383915.134}
SPL {X  -159.990, Y  +598.793, Z    +0.000, E1   -41.896, E3 +383925.888}
SPL {X  -159.990, Y  +604.215, Z    +0.000, E1   -41.919, E3 +383938.668}
SPL {X  -159.990, Y  +610.545, Z    +0.000, E1   -41.917, E3 +383953.638}
SPL {X  -159.990, Y  +615.720, Z    +0.000, E1   -41.899, E3 +383965.898}
SPL {X  -159.990, Y  +620.005, Z    +0.000, E1   -41.900, E3 +383976.031}
SPL {X  -159.990, Y  +624.919, Z    +0.000, E1   -41.912, E3 +383987.638}
SPL {X  -159.990, Y  +630.816, Z    +0.000, E1   -41.915, E3 +384001.567}
SPL {X  -159.990, Y  +637.009, Z    +0.000, E1   -41.925, E3 +384016.193}
SPL {X  -159.990, Y  +642.624, Z    +0.000, E1   -41.901, E3 +384029.514}
SPL {X  -159.990, Y  +647.782, Z    +0.000, E1   -41.914, E3 +384041.682}
SPL {X  -159.990, Y  +653.094, Z    +0.000, E1   -41.905, E3 +384054.260}
SPL {X  -159.990, Y  +657.893, Z    +0.000, E1   -41.899, E3 +384065.626}
SPL {X  -159.990, Y  +662.516, Z    +0.000, E1   -41.899, E3 +384076.557}
SPL {X  -159.990, Y  +668.411, Z    +0.000, E1   -41.929, E3 +384090.451}
SPL {X  -159.968, Y  +674.139, Z    +0.000, E1   -41.898, E3 +384104.055}
SPL {X  -159.817, Y  +678.937, Z    +0.000, E1   -41.879, E3 +384115.551}
SPL {X  -159.484, Y  +684.213, Z    +0.000, E1   -41.818, E3 +384128.387}
SPL {X  -159.007, Y  +689.209, Z    +0.000, E1   -41.732, E3 +384140.692}
SPL {X  -158.327, Y  +694.511, Z    +0.000, E1   -41.622, E3 +384153.943}
SPL {X  -157.480, Y  +699.729, Z    +0.000, E1   -41.453, E3 +384167.206}
SPL {X  -156.604, Y  +704.242, Z    +0.000, E1   -41.288, E3 +384178.815}
SPL {X  -155.514, Y  +709.078, Z    +0.000, E1   -41.107, E3 +384191.368}
SPL {X  -154.232, Y  +714.035, Z    +0.000, E1   -40.861, E3 +384204.427}
SPL {X  -153.147, Y  +717.790, Z    +0.000, E1   -40.640, E3 +384214.446}
SPL {X  -151.881, Y  +721.788, Z    +0.000, E1   -40.435, E3 +384225.132}
SPL {X  -148.572, Y  +730.857, Z    +0.000, E1   -36.304, E3 +384281.341}
ENDSPLINE

SPLINE
SPL {X  -154.420, Y  +713.347, Z    +0.000, E1   -25.698, E3 +384326.765}
SPL {X  -156.970, Y  +702.437, Z    +0.000, E1   -20.224, E3 +384338.461}
SPL {X  -159.301, Y  +686.331, Z    +0.000, E1   -11.648, E3 +384348.234}
SPL {X  -159.936, Y  +675.651, Z    +0.000, E1    -5.377, E3 +384351.950}
SPL {X  -159.990, Y  +670.142, Z    +0.000, E1    -1.740, E3 +384353.249}
SPL {X  -159.990, Y  +666.629, Z    +0.000, E1    +0.827, E3 +384353.899}
SPL {X  -159.990, Y  +662.407, Z    +0.000, E1    +4.406, E3 +384354.749}
SPL {X  -159.990, Y  +655.884, Z    +0.000, E1   +10.601, E3 +384356.615}
SPL {X  -159.990, Y  +646.242, Z    +0.000, E1   +19.956, E3 +384360.534}
SPL {X  -159.990, Y  +624.365, Z    +0.000, E1   +33.860, E3 +384378.435}
SPL {X  -159.990, Y  +615.596, Z    +0.000, E1   +36.980, E3 +384388.094}
SPL {X  -159.990, Y  +586.905, Z    +0.000, E1   +41.264, E3 +384435.120}
SPL {X  -159.990, Y  +581.111, Z    +0.000, E1   +41.245, E3 +384449.174}
SPL {X  -159.990, Y  +576.269, Z    +0.000, E1   +41.239, E3 +384460.902}
SPL {X  -159.990, Y  +571.714, Z    +0.000, E1   +41.240, E3 +384471.930}
SPL {X  -159.990, Y  +567.050, Z    +0.000, E1   +41.238, E3 +384483.217}
SPL {X  -159.990, Y  +561.959, Z    +0.000, E1   +41.251, E3 +384495.515}
SPL {X  -159.990, Y  +555.553, Z    +0.000, E1   +41.273, E3 +384510.983}
SPL {X  -159.990, Y  +548.812, Z    +0.000, E1   +41.263, E3 +384527.307}
SPL {X  -159.990, Y  +542.097, Z    +0.000, E1   +41.274, E3 +384543.560}
SPL {X  -159.990, Y  +535.325, Z    +0.000, E1   +41.260, E3 +384559.961}
SPL {X  -159.990, Y  +529.136, Z    +0.000, E1   +41.262, E3 +384574.928}
SPL {X  -159.990, Y  +522.690, Z    +0.000, E1   +41.265, E3 +384590.528}
SPL {X  -159.990, Y  +516.698, Z    +0.000, E1   +41.259, E3 +384605.002}
SPL {X  -159.990, Y  +510.896, Z    +0.000, E1   +41.267, E3 +384619.020}
SPL {X  -159.990, Y  +505.215, Z    +0.000, E1   +41.261, E3 +384632.780}
SPL {X  -159.990, Y  +498.837, Z    +0.000, E1   +41.283, E3 +384648.169}
SPL {X  -159.990, Y  +493.848, Z    +0.000, E1   +41.241, E3 +384660.289}
SPL {X  -159.990, Y  +479.011, Z    +0.000, E1   +45.740, E3 +384666.794}
SPL {X  -159.990, Y  +471.379, Z    +0.000, E1   +46.435, E3 +384678.410}
SPL {X  -159.990, Y  +466.895, Z    +0.000, E1   +45.533, E3 +384692.814}
SPL {X  -159.990, Y  +462.409, Z    +0.000, E1   +44.664, E3 +384707.589}
SPL {X  -159.990, Y  +458.229, Z    +0.000, E1   +43.579, E3 +384723.072}
ENDSPLINE

SPLINE
SPL {X  -159.990, Y  +471.362, Z    +0.000, E1   +35.782, E3 +384736.345}
ENDSPLINE

SPLINE
SPL {X  -159.990, Y  +466.474, Z    +0.000, E1   +35.796, E3 +384750.741}
SPL {X  -159.990, Y  +461.990, Z    +0.000, E1   +35.776, E3 +384763.976}
SPL {X  -159.990, Y  +457.385, Z    +0.000, E1   +35.788, E3 +384777.523}
SPL {X  -159.990, Y  +452.637, Z    +0.000, E1   +35.783, E3 +384791.515}
SPL {X  -159.990, Y  +448.227, Z    +0.000, E1   +35.776, E3 +384804.511}
SPL {X  -159.990, Y  +443.707, Z    +0.000, E1   +35.784, E3 +384817.806}
SPL {X  -159.990, Y  +439.109, Z    +0.000, E1   +35.781, E3 +384831.342}
SPL {X  -159.990, Y  +434.400, Z    +0.000, E1   +35.789, E3 +384845.197}
SPL {X  -159.990, Y  +430.115, Z    +0.000, E1   +35.777, E3 +384857.814}
SPL {X  -159.990, Y  +426.641, Z    +0.000, E1   +35.769, E3 +384868.065}
SPL {X  -159.990, Y  +422.627, Z    +0.000, E1   +35.788, E3 +384879.862}
SPL {X  -159.990, Y  +417.866, Z    +0.000, E1   +35.788, E3 +384893.876}
SPL {X  -159.990, Y  +413.498, Z    +0.000, E1   +35.779, E3 +384906.758}
SPL {X  -159.990, Y  +408.600, Z    +0.000, E1   +35.802, E3 +384921.145}
SPL {X  -159.990, Y  +403.496, Z    +0.000, E1   +35.787, E3 +384936.200}
SPL {X  -159.990, Y  +398.606, Z    +0.000, E1   +35.794, E3 +384950.588}
SPL {X  -159.990, Y  +394.138, Z    +0.000, E1   +35.778, E3 +384963.771}
SPL {X  -159.990, Y  +390.065, Z    +0.000, E1   +35.780, E3 +384975.761}
SPL {X  -159.990, Y  +385.506, Z    +0.000, E1   +35.789, E3 +384989.167}
SPL {X  -159.976, Y  +380.359, Z    +0.000, E1   +35.797, E3 +385004.316}
SPL {X  -159.831, Y  +375.358, Z    +0.000, E1   +35.763, E3 +385019.206}
SPL {X  -159.547, Y  +370.604, Z    +0.000, E1   +35.724, E3 +385033.505}
SPL {X  -159.134, Y  +365.969, Z    +0.000, E1   +35.644, E3 +385047.591}
SPL {X  -158.606, Y  +361.498, Z    +0.000, E1   +35.550, E3 +385061.355}
SPL {X  -157.918, Y  +356.833, Z    +0.000, E1   +35.439, E3 +385075.808}
SPL {X  -157.185, Y  +352.671, Z    +0.000, E1   +35.292, E3 +385088.869}
SPL {X  -156.302, Y  +348.345, Z    +0.000, E1   +35.165, E3 +385102.490}
SPL {X  -155.054, Y  +343.066, Z    +0.000, E1   +34.964, E3 +385119.304}
SPL {X  -154.305, Y  +340.232, Z    +0.000, E1   +28.975, E3 +385176.864}
ENDSPLINE

SPLINE
SPL {X  -158.456, Y  +360.399, Z    +0.000, E1   +16.490, E3 +385213.684}
SPL {X  -159.553, Y  +370.677, Z    +0.000, E1   +10.576, E3 +385221.444}
SPL {X  -159.960, Y  +379.402, Z    +0.000, E1    +5.303, E3 +385225.464}
SPL {X  -159.990, Y  +385.983, Z    +0.000, E1    +0.882, E3 +385227.537}
SPL {X  -159.990, Y  +390.933, Z    +0.000, E1    -2.877, E3 +385228.985}
SPL {X  -159.990, Y  +396.375, Z    +0.000, E1    -7.538, E3 +385230.759}
SPL {X  -159.990, Y  +404.277, Z    +0.000, E1   -14.543, E3 +385234.422}
SPL {X  -159.990, Y  +423.101, Z    +0.000, E1   -27.351, E3 +385250.861}
SPL {X  -159.990, Y  +430.933, Z    +0.000, E1   -30.672, E3 +385260.832}
SPL {X  -159.990, Y  +452.779, Z    +0.000, E1   -35.077, E3 +385302.995}
SPL {X  -159.990, Y  +457.209, Z    +0.000, E1   -35.039, E3 +385316.455}
SPL {X  -159.990, Y  +460.708, Z    +0.000, E1   -35.045, E3 +385327.037}
SPL {X  -159.990, Y  +465.240, Z    +0.000, E1   -35.066, E3 +385340.713}
SPL {X  -159.990, Y  +470.278, Z    +0.000, E1   -35.063, E3 +385355.946}
SPL {X  -159.990, Y  +474.610, Z    +0.000, E1   -35.053, E3 +385369.045}
SPL {X  -159.990, Y  +478.303, Z    +0.000, E1   -35.049, E3 +385380.217}
SPL {X  -159.990, Y  +482.537, Z    +0.000, E1   -35.066, E3 +385393.009}
SPL {X  -159.990, Y  +487.181, Z    +0.000, E1   -35.054, E3 +385407.091}
SPL {X  -159.990, Y  +492.368, Z    +0.000, E1   -35.076, E3 +385422.763}
SPL {X  -159.990, Y  +497.072, Z    +0.000, E1   -35.040, E3 +385437.060}
SPL {X  -159.990, Y  +501.645, Z    +0.000, E1   -35.067, E3 +385450.843}
SPL {X  -159.990, Y  +507.359, Z    +0.000, E1   -35.080, E3 +385468.099}
SPL {X  -159.990, Y  +513.555, Z    +0.000, E1   -35.089, E3 +385486.830}
SPL {X  -159.990, Y  +518.055, Z    +0.000, E1   -35.037, E3 +385500.516}
SPL {X  -159.990, Y  +521.637, Z    +0.000, E1   -35.056, E3 +385511.326}
SPL {X  -159.990, Y  +526.246, Z    +0.000, E1   -35.065, E3 +385525.230}
SPL {X  -159.990, Y  +531.319, Z    +0.000, E1   -35.072, E3 +385540.586}
SPL {X  -159.990, Y  +537.053, Z    +0.000, E1   -35.083, E3 +385557.918}
SPL {X  -159.990, Y  +542.114, Z    +0.000, E1   -35.053, E3 +385573.265}
SPL {X  -159.990, Y  +545.724, Z    +0.000, E1   -35.043, E3 +385584.190}
SPL {X  -159.990, Y  +549.546, Z    +0.000, E1   -35.061, E3 +385595.714}
SPL {X  -159.990, Y  +554.793, Z    +0.000, E1   -35.100, E3 +385611.477}
SPL {X  -159.990, Y  +560.931, Z    +0.000, E1   -35.098, E3 +385630.039}
SPL {X  -159.990, Y  +566.542, Z    +0.000, E1   -35.080, E3 +385647.046}
SPL {X  -159.990, Y  +571.374, Z    +0.000, E1   -35.070, E3 +385661.670}
SPL {X  -159.990, Y  +575.771, Z    +0.000, E1   -35.064, E3 +385674.975}
SPL {X  -159.990, Y  +579.185, Z    +0.000, E1   -35.047, E3 +385685.324}
SPL {X  -159.990, Y  +581.944, Z    +0.000, E1   -35.051, E3 +385693.662}
SPL {X  -159.990, Y  +585.414, Z    +0.000, E1   -35.059, E3 +385704.144}
SPL {X  -159.990, Y  +590.166, Z    +0.000, E1   -35.084, E3 +385718.473}
SPL {X  -159.990, Y  +595.313, Z    +0.000, E1   -35.073, E3 +385734.051}
SPL {X  -159.990, Y  +600.543, Z    +0.000, E1   -35.091, E3 +385749.834}
SPL {X  -159.990, Y  +605.846, Z    +0.000, E1   -35.077, E3 +385765.885}
SPL {X  -159.990, Y  +611.113, Z    +0.000, E1   -35.087, E3 +385781.791}
SPL {X  -159.990, Y  +616.690, Z    +0.000, E1   -35.089, E3 +385798.654}
SPL {X  -159.990, Y  +621.534, Z    +0.000, E1   -35.068, E3 +385813.313}
SPL {X  -159.990, Y  +625.237, Z    +0.000, E1   -35.062, E3 +385824.515}
SPL {X  -159.990, Y  +629.217, Z    +0.000, E1   -35.065, E3 +385836.573}
SPL {X  -159.990, Y  +632.566, Z    +0.000, E1   -35.044, E3 +385846.735}
SPL {X  -159.990, Y  +635.965, Z    +0.000, E1   -35.065, E3 +385856.979}
SPL {X  -159.990, Y  +640.633, Z    +0.000, E1   -35.080, E3 +385871.067}
SPL {X  -159.990, Y  +645.423, Z    +0.000, E1   -35.070, E3 +385885.573}
SPL {X  -159.990, Y  +650.555, Z    +0.000, E1   -35.089, E3 +385901.062}
SPL {X  -159.990, Y  +656.270, Z    +0.000, E1   -35.087, E3 +385918.355}
SPL {X  -159.990, Y  +661.105, Z    +0.000, E1   -35.059, E3 +385933.018}
SPL {X  -159.990, Y  +665.311, Z    +0.000, E1   -35.064, E3 +385945.733}
SPL {X  -159.990, Y  +670.193, Z    +0.000, E1   -35.076, E3 +385960.480}
SPL {X  -159.948, Y  +675.148, Z    +0.000, E1   -35.069, E3 +385975.472}
SPL {X  -159.752, Y  +680.228, Z    +0.000, E1   -35.050, E3 +385991.020}
SPL {X  -159.371, Y  +685.563, Z    +0.000, E1   -34.989, E3 +386007.532}
SPL {X  -158.886, Y  +690.264, Z    +0.000, E1   -34.888, E3 +386022.283}
SPL {X  -158.362, Y  +694.266, Z    +0.000, E1   -34.794, E3 +386034.957}
SPL {X  -157.614, Y  +698.973, Z    +0.000, E1   -34.690, E3 +386049.957}
SPL {X  -156.901, Y  +702.787, Z    +0.000, E1   -34.523, E3 +386062.301}
SPL {X  -156.097, Y  +706.580, Z    +0.000, E1   -34.427, E3 +386074.540}
SPL {X  -155.080, Y  +710.833, Z    +0.000, E1   -34.231, E3 +386088.474}
SPL {X  -153.755, Y  +715.731, Z    +0.000, E1   -30.246, E3 +386137.740}
ENDSPLINE

SPLINE
SPL {X  -155.537, Y  +708.983, Z    +0.000, E1   -25.008, E3 +386163.567}
SPL {X  -158.838, Y  +690.666, Z    +0.000, E1   -14.584, E3 +386188.280}
SPL {X  -159.750, Y  +680.262, Z    +0.000, E1    -8.563, E3 +386194.420}
SPL {X  -159.973, Y  +673.798, Z    +0.000, E1    -4.600, E3 +386196.884}
SPL {X  -159.990, Y  +668.863, Z    +0.000, E1    -1.298, E3 +386198.323}
SPL {X  -159.990, Y  +663.839, Z    +0.000, E1    +2.454, E3 +386199.584}
SPL {X  -159.990, Y  +657.071, Z    +0.000, E1    +8.297, E3 +386201.777}
SPL {X  -159.990, Y  +646.193, Z    +0.000, E1   +17.980, E3 +386207.503}
SPL {X  -159.990, Y  +621.124, Z    +0.000, E1   +32.598, E3 +386230.990}
SPL {X  -159.990, Y  +597.855, Z    +0.000, E1   +36.862, E3 +386273.910}
SPL {X  -159.990, Y  +592.884, Z    +0.000, E1   +36.865, E3 +386287.981}
SPL {X  -159.990, Y  +587.104, Z    +0.000, E1   +36.878, E3 +386304.337}
SPL {X  -159.990, Y  +581.795, Z    +0.000, E1   +36.847, E3 +386319.436}
SPL {X  -159.990, Y  +577.286, Z    +0.000, E1   +36.853, E3 +386332.193}
SPL {X  -159.990, Y  +572.409, Z    +0.000, E1   +36.854, E3 +386346.005}
SPL {X  -159.990, Y  +567.110, Z    +0.000, E1   +36.868, E3 +386360.967}
SPL {X  -159.990, Y  +562.387, Z    +0.000, E1   +36.853, E3 +386374.328}
SPL {X  -159.990, Y  +557.944, Z    +0.000, E1   +36.859, E3 +386386.922}
SPL {X  -159.990, Y  +553.661, Z    +0.000, E1   +36.844, E3 +386399.085}
SPL {X  -159.990, Y  +549.195, Z    +0.000, E1   +36.856, E3 +386411.720}
SPL {X  -159.990, Y  +544.733, Z    +0.000, E1   +36.845, E3 +386424.366}
SPL {X  -159.990, Y  +539.889, Z    +0.000, E1   +36.872, E3 +386438.051}
SPL {X  -159.990, Y  +534.469, Z    +0.000, E1   +36.855, E3 +386453.448}
SPL {X  -159.990, Y  +530.428, Z    +0.000, E1   +36.821, E3 +386464.982}
SPL {X  -159.990, Y  +525.940, Z    +0.000, E1   +36.859, E3 +386477.628}
SPL {X  -159.990, Y  +520.301, Z    +0.000, E1   +36.855, E3 +386493.605}
SPL {X  -159.990, Y  +514.308, Z    +0.000, E1   +36.869, E3 +386510.567}
SPL {X  -159.990, Y  +508.591, Z    +0.000, E1   +36.846, E3 +386526.802}
SPL {X  -159.990, Y  +503.454, Z    +0.000, E1   +36.847, E3 +386541.357}
SPL {X  -159.990, Y  +498.507, Z    +0.000, E1   +36.487, E3 +386557.806}
ENDSPLINE

SPLINE
SPL {X  -159.990, Y  +506.994, Z    +0.000, E1   +30.162, E3 +386570.315}
ENDSPLINE

SPLINE
SPL {X  -159.990, Y  +502.084, Z    +0.000, E1   +31.057, E3 +386581.966}
SPL {X  -159.990, Y  +494.586, Z    +0.000, E1   +32.444, E3 +386598.570}
SPL {X  -159.990, Y  +487.723, Z    +0.000, E1   +33.658, E3 +386613.022}
SPL {X  -159.990, Y  +481.374, Z    +0.000, E1   +34.706, E3 +386626.226}
SPL {X  -159.990, Y  +475.503, Z    +0.000, E1   +35.597, E3 +386638.279}
SPL {X  -159.990, Y  +471.459, Z    +0.000, E1   +35.779, E3 +386649.125}
SPL {X  -159.990, Y  +467.485, Z    +0.000, E1   +35.768, E3 +386660.855}
SPL {X  -159.990, Y  +462.739, Z    +0.000, E1   +35.799, E3 +386674.783}
SPL {X  -159.990, Y  +457.385, Z    +0.000, E1   +35.788, E3 +386690.566}
SPL {X  -159.990, Y  +452.637, Z    +0.000, E1   +35.783, E3 +386704.558}
SPL {X  -159.990, Y  +448.227, Z    +0.000, E1   +35.776, E3 +386717.555}
SPL {X  -159.990, Y  +443.707, Z    +0.000, E1   +35.784, E3 +386730.850}
SPL {X  -159.990, Y  +439.109, Z    +0.000, E1   +35.781, E3 +386744.386}
SPL {X  -159.990, Y  +434.400, Z    +0.000, E1   +35.789, E3 +386758.241}
SPL {X  -159.990, Y  +430.115, Z    +0.000, E1   +35.777, E3 +386770.858}
SPL {X  -159.990, Y  +425.407, Z    +0.000, E1   +35.800, E3 +386784.697}
SPL {X  -159.990, Y  +420.199, Z    +0.000, E1   +35.790, E3 +386800.052}
SPL {X  -159.990, Y  +414.514, Z    +0.000, E1   +35.815, E3 +386816.750}
SPL {X  -159.990, Y  +409.702, Z    +0.000, E1   +35.772, E3 +386830.991}
SPL {X  -159.990, Y  +405.848, Z    +0.000, E1   +35.776, E3 +386842.337}
SPL {X  -159.990, Y  +400.924, Z    +0.000, E1   +35.804, E3 +386856.795}
SPL {X  -159.990, Y  +395.017, Z    +0.000, E1   +35.806, E3 +386874.184}
SPL {X  -159.990, Y  +390.065, Z    +0.000, E1   +35.780, E3 +386888.805}
SPL {X  -159.990, Y  +385.506, Z    +0.000, E1   +35.789, E3 +386902.210}
SPL {X  -159.976, Y  +380.359, Z    +0.000, E1   +35.797, E3 +386917.359}
SPL {X  -159.831, Y  +375.358, Z    +0.000, E1   +35.763, E3 +386932.249}
SPL {X  -159.547, Y  +370.604, Z    +0.000, E1   +35.724, E3 +386946.549}
SPL {X  -159.134, Y  +365.969, Z    +0.000, E1   +35.644, E3 +386960.634}
SPL {X  -158.715, Y  +362.338, Z    +0.000, E1   +35.547, E3 +386971.842}
SPL {X  -158.237, Y  +358.884, Z    +0.000, E1   +35.480, E3 +386982.499}
SPL {X  -157.724, Y  +355.670, Z    +0.000, E1   +35.371, E3 +386992.533}
SPL {X  -157.185, Y  +352.671, Z    +0.000, E1   +35.292, E3 +387001.912}
SPL {X  -156.582, Y  +349.653, Z    +0.000, E1   +35.175, E3 +387011.445}
SPL {X  -155.743, Y  +345.880, Z    +0.000, E1   +35.068, E3 +387023.372}
SPL {X  -154.759, Y  +341.925, Z    +0.000, E1   +34.868, E3 +387036.078}
SPL {X  -154.305, Y  +340.232, Z    +0.000, E1   +28.975, E3 +387089.908}
ENDSPLINE

SPLINE
SPL {X  -158.456, Y  +360.399, Z    +0.000, E1   +16.490, E3 +387126.727}
SPL {X  -159.553, Y  +370.677, Z    +0.000, E1   +10.576, E3 +387134.488}
SPL {X  -159.960, Y  +379.402, Z    +0.000, E1    +5.303, E3 +387138.508}
SPL {X  -159.990, Y  +385.983, Z    +0.000, E1    +0.882, E3 +387140.580}
SPL {X  -159.990, Y  +390.933, Z    +0.000, E1    -2.877, E3 +387142.028}
SPL {X  -159.990, Y  +396.375, Z    +0.000, E1    -7.538, E3 +387143.803}
SPL {X  -159.990, Y  +404.277, Z    +0.000, E1   -14.543, E3 +387147.466}
SPL {X  -159.990, Y  +423.101, Z    +0.000, E1   -27.351, E3 +387163.905}
SPL {X  -159.990, Y  +430.933, Z    +0.000, E1   -30.672, E3 +387173.875}
SPL {X  -159.990, Y  +451.842, Z    +0.000, E1   -35.050, E3 +387213.247}
SPL {X  -159.990, Y  +456.402, Z    +0.000, E1   -35.061, E3 +387227.023}
SPL {X  -159.990, Y  +460.708, Z    +0.000, E1   -35.045, E3 +387240.081}
SPL {X  -159.990, Y  +465.240, Z    +0.000, E1   -35.066, E3 +387253.756}
SPL {X  -159.990, Y  +470.278, Z    +0.000, E1   -35.063, E3 +387268.990}
SPL {X  -159.990, Y  +474.610, Z    +0.000, E1   -35.053, E3 +387282.088}
SPL {X  -159.990, Y  +478.303, Z    +0.000, E1   -35.049, E3 +387293.261}
SPL {X  -159.990, Y  +482.537, Z    +0.000, E1   -35.066, E3 +387306.052}
SPL {X  -159.990, Y  +487.181, Z    +0.000, E1   -35.054, E3 +387320.135}
SPL {X  -159.990, Y  +490.807, Z    +0.000, E1   -35.036, E3 +387331.136}
SPL {X  -159.990, Y  +493.669, Z    +0.000, E1   -35.034, E3 +387339.816}
SPL {X  -159.990, Y  +497.072, Z    +0.000, E1   -35.040, E3 +387350.103}
SPL {X  -159.990, Y  +501.645, Z    +0.000, E1   -35.067, E3 +387363.886}
SPL {X  -159.990, Y  +506.307, Z    +0.000, E1   -35.049, E3 +387378.008}
SPL {X  -159.990, Y  +510.443, Z    +0.000, E1   -35.051, E3 +387390.521}
SPL {X  -159.990, Y  +514.632, Z    +0.000, E1   -35.050, E3 +387403.191}
SPL {X  -159.990, Y  +518.055, Z    +0.000, E1   -35.037, E3 +387413.560}
SPL {X  -159.990, Y  +521.637, Z    +0.000, E1   -35.056, E3 +387424.370}
SPL {X  -159.990, Y  +526.246, Z    +0.000, E1   -35.065, E3 +387438.273}
SPL {X  -159.990, Y  +530.289, Z    +0.000, E1   -35.044, E3 +387450.559}
SPL {X  -159.990, Y  +534.797, Z    +0.000, E1   -35.069, E3 +387464.160}
SPL {X  -159.990, Y  +538.710, Z    +0.000, E1   -35.033, E3 +387476.056}
SPL {X  -159.990, Y  +542.114, Z    +0.000, E1   -35.053, E3 +387486.309}
SPL {X  -159.990, Y  +545.724, Z    +0.000, E1   -35.043, E3 +387497.233}
SPL {X  -159.990, Y  +549.546, Z    +0.000, E1   -35.061, E3 +387508.757}
SPL {X  -159.990, Y  +552.868, Z    +0.000, E1   -35.047, E3 +387518.799}
SPL {X  -159.990, Y  +557.043, Z    +0.000, E1   -35.087, E3 +387531.337}
SPL {X  -159.990, Y  +561.808, Z    +0.000, E1   -35.066, E3 +387545.790}
SPL {X  -159.990, Y  +566.542, Z    +0.000, E1   -35.080, E3 +387560.090}
SPL {X  -159.990, Y  +570.261, Z    +0.000, E1   -35.046, E3 +387571.386}
SPL {X  -159.990, Y  +574.780, Z    +0.000, E1   -35.101, E3 +387584.966}
SPL {X  -159.990, Y  +579.185, Z    +0.000, E1   -35.047, E3 +387598.367}
SPL {X  -159.990, Y  +581.944, Z    +0.000, E1   -35.051, E3 +387606.705}
SPL {X  -159.990, Y  +585.414, Z    +0.000, E1   -35.059, E3 +387617.188}
SPL {X  -159.990, Y  +588.716, Z    +0.000, E1   -35.047, E3 +387627.191}
SPL {X  -159.990, Y  +592.923, Z    +0.000, E1   -35.084, E3 +387639.855}
SPL {X  -159.990, Y  +598.554, Z    +0.000, E1   -35.088, E3 +387656.874}
SPL {X  -159.990, Y  +603.289, Z    +0.000, E1   -35.068, E3 +387671.201}
SPL {X  -159.990, Y  +607.919, Z    +0.000, E1   -35.079, E3 +387685.190}
SPL {X  -159.990, Y  +613.036, Z    +0.000, E1   -35.082, E3 +387700.661}
SPL {X  -159.990, Y  +617.577, Z    +0.000, E1   -35.061, E3 +387714.423}
SPL {X  -159.990, Y  +621.534, Z    +0.000, E1   -35.068, E3 +387726.357}
SPL {X  -159.990, Y  +626.426, Z    +0.000, E1   -35.093, E3 +387741.116}
SPL {X  -159.990, Y  +631.553, Z    +0.000, E1   -35.068, E3 +387756.674}
SPL {X  -159.990, Y  +635.965, Z    +0.000, E1   -35.065, E3 +387770.022}
SPL {X  -159.990, Y  +640.633, Z    +0.000, E1   -35.080, E3 +387784.111}
SPL {X  -159.990, Y  +645.423, Z    +0.000, E1   -35.070, E3 +387798.616}
SPL {X  -159.990, Y  +650.555, Z    +0.000, E1   -35.089, E3 +387814.105}
SPL {X  -159.990, Y  +656.270, Z    +0.000, E1   -35.087, E3 +387831.398}
SPL {X  -159.990, Y  +661.105, Z    +0.000, E1   -35.059, E3 +387846.062}
SPL {X  -159.990, Y  +665.311, Z    +0.000, E1   -35.064, E3 +387858.777}
SPL {X  -159.990, Y  +670.193, Z    +0.000, E1   -35.076, E3 +387873.524}
SPL {X  -159.948, Y  +675.148, Z    +0.000, E1   -35.069, E3 +387888.516}
SPL {X  -159.805, Y  +679.202, Z    +0.000, E1   -35.029, E3 +387900.948}
SPL {X  -159.584, Y  +682.885, Z    +0.000, E1   -34.997, E3 +387912.308}
SPL {X  -159.292, Y  +686.426, Z    +0.000, E1   -34.947, E3 +387923.310}
SPL {X  -158.886, Y  +690.264, Z    +0.000, E1   -34.888, E3 +387935.326}
SPL {X  -158.362, Y  +694.266, Z    +0.000, E1   -34.794, E3 +387948.000}
SPL {X  -157.614, Y  +698.973, Z    +0.000, E1   -34.690, E3 +387963.000}
SPL {X  -156.901, Y  +702.787, Z    +0.000, E1   -34.523, E3 +387975.344}
SPL {X  -156.097, Y  +706.580, Z    +0.000, E1   -34.427, E3 +387987.584}
SPL {X  -155.080, Y  +710.833, Z    +0.000, E1   -34.231, E3 +388001.518}
SPL {X  -153.755, Y  +715.731, Z    +0.000, E1   -30.246, E3 +388050.784}
ENDSPLINE

SPLINE
SPL {X  -155.537, Y  +708.983, Z    +0.000, E1   -25.008, E3 +388076.610}
SPL {X  -158.838, Y  +690.666, Z    +0.000, E1   -14.584, E3 +388101.323}
SPL {X  -159.750, Y  +680.262, Z    +0.000, E1    -8.563, E3 +388107.464}
SPL {X  -159.973, Y  +673.798, Z    +0.000, E1    -4.600, E3 +388109.927}
SPL {X  -159.990, Y  +668.863, Z    +0.000, E1    -1.298, E3 +388111.367}
SPL {X  -159.990, Y  +663.839, Z    +0.000, E1    +2.454, E3 +388112.628}
SPL {X  -159.990, Y  +658.349, Z    +0.000, E1    +7.223, E3 +388114.310}
SPL {X  -159.990, Y  +650.390, Z    +0.000, E1   +14.372, E3 +388118.056}
SPL {X  -159.990, Y  +643.417, Z    +0.000, E1   +20.300, E3 +388122.320}
SPL {X  -159.990, Y  +621.124, Z    +0.000, E1   +32.598, E3 +388144.034}
SPL {X  -159.990, Y  +597.855, Z    +0.000, E1   +36.862, E3 +388186.953}
SPL {X  -159.990, Y  +592.884, Z    +0.000, E1   +36.865, E3 +388201.024}
SPL {X  -159.990, Y  +587.104, Z    +0.000, E1   +36.878, E3 +388217.381}
SPL {X  -159.990, Y  +581.795, Z    +0.000, E1   +36.847, E3 +388232.480}
SPL {X  -159.990, Y  +576.165, Z    +0.000, E1   +36.887, E3 +388248.359}
SPL {X  -159.990, Y  +570.328, Z    +0.000, E1   +36.855, E3 +388264.932}
SPL {X  -159.990, Y  +566.126, Z    +0.000, E1   +36.841, E3 +388276.839}
SPL {X  -159.990, Y  +562.387, Z    +0.000, E1   +36.853, E3 +388287.371}
SPL {X  -159.990, Y  +557.944, Z    +0.000, E1   +36.859, E3 +388299.965}
SPL {X  -159.990, Y  +552.571, Z    +0.000, E1   +36.873, E3 +388315.169}
SPL {X  -159.990, Y  +546.127, Z    +0.000, E1   +36.890, E3 +388333.396}
SPL {X  -159.990, Y  +539.889, Z    +0.000, E1   +36.872, E3 +388351.094}
SPL {X  -159.990, Y  +534.469, Z    +0.000, E1   +36.855, E3 +388366.492}
SPL {X  -159.990, Y  +528.569, Z    +0.000, E1   +36.871, E3 +388383.210}
SPL {X  -159.990, Y  +522.641, Z    +0.000, E1   +36.854, E3 +388400.021}
SPL {X  -159.990, Y  +517.225, Z    +0.000, E1   +36.859, E3 +388415.355}
SPL {X  -159.990, Y  +511.408, Z    +0.000, E1   +36.858, E3 +388431.843}
SPL {X  -159.990, Y  +505.756, Z    +0.000, E1   +36.857, E3 +388447.853}
SPL {X  -159.990, Y  +499.829, Z    +0.000, E1   +36.864, E3 +388464.658}
SPL {X  -159.990, Y  +498.054, Z    +0.000, E1   +35.692, E3 +388476.697}
ENDSPLINE

SPLINE
SPL {X  -159.990, Y  +506.994, Z    +0.000, E1   +30.162, E3 +388483.359}
ENDSPLINE

SPLINE
SPL {X  -159.990, Y  +502.084, Z    +0.000, E1   +31.057, E3 +388495.010}
SPL {X  -159.990, Y  +494.586, Z    +0.000, E1   +32.444, E3 +388511.613}
SPL {X  -159.990, Y  +486.073, Z    +0.000, E1   +33.960, E3 +388529.451}
SPL {X  -159.990, Y  +477.314, Z    +0.000, E1   +35.342, E3 +388547.629}
SPL {X  -159.990, Y  +471.459, Z    +0.000, E1   +35.779, E3 +388562.169}
SPL {X  -159.990, Y  +466.474, Z    +0.000, E1   +35.796, E3 +388576.828}
SPL {X  -159.990, Y  +461.990, Z    +0.000, E1   +35.776, E3 +388590.063}
SPL {X  -159.990, Y  +458.524, Z    +0.000, E1   +35.761, E3 +388600.300}
SPL {X  -159.990, Y  +453.597, Z    +0.000, E1   +35.819, E3 +388614.720}
SPL {X  -159.990, Y  +448.227, Z    +0.000, E1   +35.776, E3 +388630.598}
SPL {X  -159.990, Y  +443.707, Z    +0.000, E1   +35.784, E3 +388643.893}
SPL {X  -159.990, Y  +439.109, Z    +0.000, E1   +35.781, E3 +388657.429}
SPL {X  -159.990, Y  +435.535, Z    +0.000, E1   +35.764, E3 +388667.980}
SPL {X  -159.990, Y  +431.100, Z    +0.000, E1   +35.807, E3 +388680.965}
SPL {X  -159.990, Y  +425.407, Z    +0.000, E1   +35.800, E3 +388697.741}
SPL {X  -159.990, Y  +420.199, Z    +0.000, E1   +35.790, E3 +388713.095}
SPL {X  -159.990, Y  +414.514, Z    +0.000, E1   +35.815, E3 +388729.794}
SPL {X  -159.990, Y  +408.600, Z    +0.000, E1   +35.802, E3 +388747.232}
SPL {X  -159.990, Y  +403.496, Z    +0.000, E1   +35.787, E3 +388762.287}
SPL {X  -159.990, Y  +398.606, Z    +0.000, E1   +35.794, E3 +388776.675}
SPL {X  -159.990, Y  +394.138, Z    +0.000, E1   +35.778, E3 +388789.858}
SPL {X  -159.990, Y  +390.065, Z    +0.000, E1   +35.780, E3 +388801.848}
SPL {X  -159.990, Y  +385.506, Z    +0.000, E1   +35.789, E3 +388815.253}
SPL {X  -159.976, Y  +380.359, Z    +0.000, E1   +35.797, E3 +388830.403}
SPL {X  -159.831, Y  +375.358, Z    +0.000, E1   +35.763, E3 +388845.292}
SPL {X  -159.547, Y  +370.604, Z    +0.000, E1   +35.724, E3 +388859.592}
SPL {X  -159.134, Y  +365.969, Z    +0.000, E1   +35.644, E3 +388873.678}
SPL {X  -158.606, Y  +361.498, Z    +0.000, E1   +35.550, E3 +388887.442}
SPL {X  -157.918, Y  +356.833, Z    +0.000, E1   +35.439, E3 +388901.895}
SPL {X  -157.185, Y  +352.671, Z    +0.000, E1   +35.292, E3 +388914.956}
SPL {X  -156.302, Y  +348.345, Z    +0.000, E1   +35.165, E3 +388928.577}
SPL {X  -155.054, Y  +343.066, Z    +0.000, E1   +34.964, E3 +388945.391}
SPL {X  -154.305, Y  +340.232, Z    +0.000, E1   +28.975, E3 +389002.951}
ENDSPLINE

SPLINE
SPL {X  -158.456, Y  +360.399, Z    +0.000, E1   +16.490, E3 +389039.771}
SPL {X  -159.553, Y  +370.677, Z    +0.000, E1   +10.576, E3 +389047.531}
SPL {X  -159.960, Y  +379.402, Z    +0.000, E1    +5.303, E3 +389051.551}
SPL {X  -159.990, Y  +385.983, Z    +0.000, E1    +0.882, E3 +389053.624}
SPL {X  -159.990, Y  +390.933, Z    +0.000, E1    -2.877, E3 +389055.072}
SPL {X  -159.990, Y  +396.375, Z    +0.000, E1    -7.538, E3 +389056.846}
SPL {X  -159.990, Y  +405.219, Z    +0.000, E1   -15.296, E3 +389061.164}
SPL {X  -159.990, Y  +427.416, Z    +0.000, E1   -29.294, E3 +389082.218}
SPL {X  -159.990, Y  +447.483, Z    +0.000, E1   -34.518, E3 +389116.384}
SPL {X  -159.990, Y  +453.425, Z    +0.000, E1   -35.055, E3 +389131.067}
SPL {X  -159.990, Y  +457.209, Z    +0.000, E1   -35.039, E3 +389142.542}
SPL {X  -159.990, Y  +460.708, Z    +0.000, E1   -35.045, E3 +389153.124}
SPL {X  -159.990, Y  +464.162, Z    +0.000, E1   -35.038, E3 +389163.580}
SPL {X  -159.990, Y  +467.857, Z    +0.000, E1   -35.053, E3 +389174.737}
SPL {X  -159.990, Y  +471.326, Z    +0.000, E1   -35.038, E3 +389185.232}
SPL {X  -159.990, Y  +474.610, Z    +0.000, E1   -35.053, E3 +389195.132}
SPL {X  -159.990, Y  +478.303, Z    +0.000, E1   -35.049, E3 +389206.304}
SPL {X  -159.990, Y  +482.537, Z    +0.000, E1   -35.066, E3 +389219.096}
SPL {X  -159.990, Y  +487.181, Z    +0.000, E1   -35.054, E3 +389233.178}
SPL {X  -159.990, Y  +492.368, Z    +0.000, E1   -35.076, E3 +389248.850}
SPL {X  -159.990, Y  +497.072, Z    +0.000, E1   -35.040, E3 +389263.146}
SPL {X  -159.990, Y  +501.645, Z    +0.000, E1   -35.067, E3 +389276.930}
SPL {X  -159.990, Y  +506.307, Z    +0.000, E1   -35.049, E3 +389291.051}
SPL {X  -159.990, Y  +511.643, Z    +0.000, E1   -35.091, E3 +389307.132}
SPL {X  -159.990, Y  +517.156, Z    +0.000, E1   -35.059, E3 +389323.850}
SPL {X  -159.990, Y  +521.637, Z    +0.000, E1   -35.056, E3 +389337.413}
SPL {X  -159.990, Y  +526.246, Z    +0.000, E1   -35.065, E3 +389351.317}
SPL {X  -159.990, Y  +530.289, Z    +0.000, E1   -35.044, E3 +389363.603}
SPL {X  -159.990, Y  +534.797, Z    +0.000, E1   -35.069, E3 +389377.203}
SPL {X  -159.990, Y  +538.710, Z    +0.000, E1   -35.033, E3 +389389.100}
SPL {X  -159.990, Y  +542.114, Z    +0.000, E1   -35.053, E3 +389399.352}
SPL {X  -159.990, Y  +546.612, Z    +0.000, E1   -35.065, E3 +389412.923}
SPL {X  -159.990, Y  +551.596, Z    +0.000, E1   -35.079, E3 +389427.959}
SPL {X  -159.990, Y  +556.051, Z    +0.000, E1   -35.060, E3 +389441.421}
SPL {X  -159.990, Y  +560.931, Z    +0.000, E1   -35.098, E3 +389456.126}
SPL {X  -159.990, Y  +564.815, Z    +0.000, E1   -35.041, E3 +389467.974}
SPL {X  -159.990, Y  +567.494, Z    +0.000, E1   -35.052, E3 +389476.054}
SPL {X  -159.990, Y  +571.374, Z    +0.000, E1   -35.070, E3 +389487.757}
SPL {X  -159.990, Y  +575.771, Z    +0.000, E1   -35.064, E3 +389501.062}
SPL {X  -159.990, Y  +580.750, Z    +0.000, E1   -35.087, E3 +389516.085}
SPL {X  -159.990, Y  +585.414, Z    +0.000, E1   -35.059, E3 +389530.231}
SPL {X  -159.990, Y  +590.166, Z    +0.000, E1   -35.084, E3 +389544.560}
SPL {X  -159.990, Y  +595.313, Z    +0.000, E1   -35.073, E3 +389560.138}
SPL {X  -159.990, Y  +599.479, Z    +0.000, E1   -35.059, E3 +389572.756}
SPL {X  -159.990, Y  +603.289, Z    +0.000, E1   -35.068, E3 +389584.245}
SPL {X  -159.990, Y  +607.919, Z    +0.000, E1   -35.079, E3 +389598.234}
SPL {X  -159.990, Y  +613.036, Z    +0.000, E1   -35.082, E3 +389613.704}
SPL {X  -159.990, Y  +617.577, Z    +0.000, E1   -35.061, E3 +389627.466}
SPL {X  -159.990, Y  +621.534, Z    +0.000, E1   -35.068, E3 +389639.400}
SPL {X  -159.990, Y  +626.426, Z    +0.000, E1   -35.093, E3 +389654.160}
SPL {X  -159.990, Y  +631.553, Z    +0.000, E1   -35.068, E3 +389669.718}
SPL {X  -159.990, Y  +635.965, Z    +0.000, E1   -35.065, E3 +389683.066}
SPL {X  -159.990, Y  +640.633, Z    +0.000, E1   -35.080, E3 +389697.154}
SPL {X  -159.990, Y  +645.423, Z    +0.000, E1   -35.070, E3 +389711.660}
SPL {X  -159.990, Y  +650.555, Z    +0.000, E1   -35.089, E3 +389727.149}
SPL {X  -159.990, Y  +656.270, Z    +0.000, E1   -35.087, E3 +389744.442}
SPL {X  -159.990, Y  +661.105, Z    +0.000, E1   -35.059, E3 +389759.105}
SPL {X  -159.990, Y  +665.311, Z    +0.000, E1   -35.064, E3 +389771.820}
SPL {X  -159.990, Y  +670.193, Z    +0.000, E1   -35.076, E3 +389786.567}
SPL {X  -159.948, Y  +675.148, Z    +0.000, E1   -35.069, E3 +389801.559}
SPL {X  -159.752, Y  +680.228, Z    +0.000, E1   -35.050, E3 +389817.107}
SPL {X  -159.371, Y  +685.563, Z    +0.000, E1   -34.989, E3 +389833.619}
SPL {X  -158.886, Y  +690.264, Z    +0.000, E1   -34.888, E3 +389848.370}
SPL {X  -158.362, Y  +694.266, Z    +0.000, E1   -34.794, E3 +389861.044}
SPL {X  -157.614, Y  +698.973, Z    +0.000, E1   -34.690, E3 +389876.044}
SPL {X  -156.640, Y  +704.066, Z    +0.000, E1   -34.516, E3 +389892.469}
SPL {X  -155.835, Y  +707.723, Z    +0.000, E1   -34.344, E3 +389904.411}
SPL {X  -155.153, Y  +710.542, Z    +0.000, E1   -34.234, E3 +389913.631}
SPL {X  -153.767, Y  +715.686, Z    +0.000, E1   -30.747, E3 +389958.849}
ENDSPLINE

SPLINE
SPL {X  -154.589, Y  +712.719, Z    +0.000, E1   -27.400, E3 +389980.249}
SPL {X  -158.529, Y  +693.075, Z    +0.000, E1   -15.996, E3 +390012.096}
SPL {X  -159.750, Y  +680.262, Z    +0.000, E1    -8.563, E3 +390020.507}
SPL {X  -159.973, Y  +673.798, Z    +0.000, E1    -4.600, E3 +390022.971}
SPL {X  -159.990, Y  +667.448, Z    +0.000, E1    -0.356, E3 +390024.751}
SPL {X  -159.990, Y  +662.686, Z    +0.000, E1    +3.472, E3 +390025.985}
SPL {X  -159.990, Y  +658.349, Z    +0.000, E1    +7.223, E3 +390027.353}
SPL {X  -159.990, Y  +653.910, Z    +0.000, E1   +11.344, E3 +390029.121}
SPL {X  -159.990, Y  +646.193, Z    +0.000, E1   +17.980, E3 +390033.590}
SPL {X  -159.990, Y  +621.124, Z    +0.000, E1   +32.598, E3 +390057.077}
SPL {X  -159.990, Y  +599.888, Z    +0.000, E1   +36.828, E3 +390094.317}
SPL {X  -159.990, Y  +595.346, Z    +0.000, E1   +36.880, E3 +390107.083}
SPL {X  -159.990, Y  +589.749, Z    +0.000, E1   +36.860, E3 +390122.956}
SPL {X  -159.990, Y  +585.754, Z    +0.000, E1   +36.838, E3 +390134.311}
SPL {X  -159.990, Y  +581.795, Z    +0.000, E1   +36.847, E3 +390145.523}
SPL {X  -159.990, Y  +576.165, Z    +0.000, E1   +36.887, E3 +390161.403}
SPL {X  -159.990, Y  +570.328, Z    +0.000, E1   +36.855, E3 +390177.976}
SPL {X  -159.990, Y  +566.126, Z    +0.000, E1   +36.841, E3 +390189.882}
SPL {X  -159.990, Y  +562.387, Z    +0.000, E1   +36.853, E3 +390200.415}
SPL {X  -159.990, Y  +557.944, Z    +0.000, E1   +36.859, E3 +390213.008}
SPL {X  -159.990, Y  +552.571, Z    +0.000, E1   +36.873, E3 +390228.213}
SPL {X  -159.990, Y  +548.223, Z    +0.000, E1   +36.832, E3 +390240.603}
SPL {X  -159.990, Y  +543.458, Z    +0.000, E1   +36.882, E3 +390254.006}
SPL {X  -159.990, Y  +537.639, Z    +0.000, E1   +36.860, E3 +390270.543}
SPL {X  -159.990, Y  +531.894, Z    +0.000, E1   +36.865, E3 +390286.832}
SPL {X  -159.990, Y  +525.940, Z    +0.000, E1   +36.859, E3 +390303.715}
SPL {X  -159.990, Y  +520.301, Z    +0.000, E1   +36.855, E3 +390319.692}
SPL {X  -159.990, Y  +516.005, Z    +0.000, E1   +36.824, E3 +390331.918}
SPL {X  -159.990, Y  +511.408, Z    +0.000, E1   +36.858, E3 +390344.887}
SPL {X  -159.990, Y  +505.756, Z    +0.000, E1   +36.857, E3 +390360.897}
SPL {X  -159.990, Y  +499.829, Z    +0.000, E1   +36.864, E3 +390377.701}
SPL {X  -159.990, Y  +498.054, Z    +0.000, E1   +35.692, E3 +390389.741}
ENDSPLINE

SPLINE
SPL {X  -159.990, Y  +506.994, Z    +0.000, E1   +30.162, E3 +390396.402}
ENDSPLINE

SPLINE
SPL {X  -159.990, Y  +502.084, Z    +0.000, E1   +31.057, E3 +390408.053}
SPL {X  -159.990, Y  +494.586, Z    +0.000, E1   +32.444, E3 +390424.657}
SPL {X  -159.990, Y  +487.723, Z    +0.000, E1   +33.658, E3 +390439.109}
SPL {X  -159.990, Y  +481.374, Z    +0.000, E1   +34.706, E3 +390452.313}
SPL {X  -159.990, Y  +475.503, Z    +0.000, E1   +35.597, E3 +390464.366}
SPL {X  -159.990, Y  +471.459, Z    +0.000, E1   +35.779, E3 +390475.212}
SPL {X  -159.990, Y  +466.474, Z    +0.000, E1   +35.796, E3 +390489.871}
SPL {X  -159.990, Y  +461.990, Z    +0.000, E1   +35.776, E3 +390503.106}
SPL {X  -159.990, Y  +457.385, Z    +0.000, E1   +35.788, E3 +390516.653}
SPL {X  -159.990, Y  +452.637, Z    +0.000, E1   +35.783, E3 +390530.645}
SPL {X  -159.990, Y  +446.982, Z    +0.000, E1   +35.815, E3 +390547.247}
SPL {X  -159.990, Y  +442.593, Z    +0.000, E1   +35.759, E3 +390560.256}
SPL {X  -159.990, Y  +439.109, Z    +0.000, E1   +35.781, E3 +390570.473}
SPL {X  -159.990, Y  +435.535, Z    +0.000, E1   +35.764, E3 +390581.023}
SPL {X  -159.990, Y  +431.100, Z    +0.000, E1   +35.807, E3 +390594.009}
SPL {X  -159.990, Y  +426.641, Z    +0.000, E1   +35.769, E3 +390607.195}
SPL {X  -159.990, Y  +422.627, Z    +0.000, E1   +35.788, E3 +390618.993}
SPL {X  -159.990, Y  +417.866, Z    +0.000, E1   +35.788, E3 +390633.006}
SPL {X  -159.990, Y  +413.498, Z    +0.000, E1   +35.779, E3 +390645.888}
SPL {X  -159.990, Y  +408.600, Z    +0.000, E1   +35.802, E3 +390660.276}
SPL {X  -159.990, Y  +403.496, Z    +0.000, E1   +35.787, E3 +390675.331}
SPL {X  -159.990, Y  +398.606, Z    +0.000, E1   +35.794, E3 +390689.718}
SPL {X  -159.990, Y  +394.138, Z    +0.000, E1   +35.778, E3 +390702.901}
SPL {X  -159.990, Y  +390.065, Z    +0.000, E1   +35.780, E3 +390714.891}
SPL {X  -159.990, Y  +385.506, Z    +0.000, E1   +35.789, E3 +390728.297}
SPL {X  -159.976, Y  +380.359, Z    +0.000, E1   +35.797, E3 +390743.446}
SPL {X  -159.831, Y  +375.358, Z    +0.000, E1   +35.763, E3 +390758.336}
SPL {X  -159.547, Y  +370.604, Z    +0.000, E1   +35.724, E3 +390772.636}
SPL {X  -159.134, Y  +365.969, Z    +0.000, E1   +35.644, E3 +390786.721}
SPL {X  -158.606, Y  +361.498, Z    +0.000, E1   +35.550, E3 +390800.485}
SPL {X  -157.918, Y  +356.833, Z    +0.000, E1   +35.439, E3 +390814.938}
SPL {X  -157.185, Y  +352.671, Z    +0.000, E1   +35.292, E3 +390827.999}
SPL {X  -156.582, Y  +349.653, Z    +0.000, E1   +35.175, E3 +390837.532}
SPL {X  -155.743, Y  +345.880, Z    +0.000, E1   +35.068, E3 +390849.459}
SPL {X  -154.759, Y  +341.925, Z    +0.000, E1   +34.868, E3 +390862.165}
SPL {X  -154.305, Y  +340.232, Z    +0.000, E1   +28.975, E3 +390915.995}
ENDSPLINE

SPLINE
SPL {X  -158.456, Y  +360.399, Z    +0.000, E1   +16.490, E3 +390952.814}
SPL {X  -159.553, Y  +370.677, Z    +0.000, E1   +10.576, E3 +390960.574}
SPL {X  -159.960, Y  +379.402, Z    +0.000, E1    +5.303, E3 +390964.595}
SPL {X  -159.990, Y  +387.301, Z    +0.000, E1    +0.001, E3 +390967.056}
SPL {X  -159.990, Y  +392.161, Z    +0.000, E1    -3.946, E3 +390968.467}
SPL {X  -159.990, Y  +396.375, Z    +0.000, E1    -7.538, E3 +390969.890}
SPL {X  -159.990, Y  +405.219, Z    +0.000, E1   -15.296, E3 +390974.207}
SPL {X  -159.990, Y  +427.882, Z    +0.000, E1   -29.477, E3 +390995.887}
SPL {X  -159.990, Y  +452.779, Z    +0.000, E1   -35.077, E3 +391042.126}
SPL {X  -159.990, Y  +457.209, Z    +0.000, E1   -35.039, E3 +391055.585}
SPL {X  -159.990, Y  +460.708, Z    +0.000, E1   -35.045, E3 +391066.168}
SPL {X  -159.990, Y  +465.240, Z    +0.000, E1   -35.066, E3 +391079.843}
SPL {X  -159.990, Y  +470.278, Z    +0.000, E1   -35.063, E3 +391095.077}
SPL {X  -159.990, Y  +474.610, Z    +0.000, E1   -35.053, E3 +391108.175}
SPL {X  -159.990, Y  +478.303, Z    +0.000, E1   -35.049, E3 +391119.348}
SPL {X  -159.990, Y  +482.537, Z    +0.000, E1   -35.066, E3 +391132.139}
SPL {X  -159.990, Y  +487.181, Z    +0.000, E1   -35.054, E3 +391146.222}
SPL {X  -159.990, Y  +492.368, Z    +0.000, E1   -35.076, E3 +391161.894}
SPL {X  -159.990, Y  +497.072, Z    +0.000, E1   -35.040, E3 +391176.190}
SPL {X  -159.990, Y  +501.645, Z    +0.000, E1   -35.067, E3 +391189.973}
SPL {X  -159.990, Y  +506.307, Z    +0.000, E1   -35.049, E3 +391204.095}
SPL {X  -159.990, Y  +510.443, Z    +0.000, E1   -35.051, E3 +391216.608}
SPL {X  -159.990, Y  +514.632, Z    +0.000, E1   -35.050, E3 +391229.278}
SPL {X  -159.990, Y  +518.055, Z    +0.000, E1   -35.037, E3 +391239.647}
SPL {X  -159.990, Y  +521.637, Z    +0.000, E1   -35.056, E3 +391250.457}
SPL {X  -159.990, Y  +526.246, Z    +0.000, E1   -35.065, E3 +391264.360}
SPL {X  -159.990, Y  +530.289, Z    +0.000, E1   -35.044, E3 +391276.646}
SPL {X  -159.990, Y  +534.797, Z    +0.000, E1   -35.069, E3 +391290.246}
SPL {X  -159.990, Y  +538.710, Z    +0.000, E1   -35.033, E3 +391302.143}
SPL {X  -159.990, Y  +542.114, Z    +0.000, E1   -35.053, E3 +391312.395}
SPL {X  -159.990, Y  +546.612, Z    +0.000, E1   -35.065, E3 +391325.967}
SPL {X  -159.990, Y  +551.596, Z    +0.000, E1   -35.079, E3 +391341.002}
SPL {X  -159.990, Y  +557.043, Z    +0.000, E1   -35.087, E3 +391357.424}
SPL {X  -159.990, Y  +562.842, Z    +0.000, E1   -35.098, E3 +391374.956}
SPL {X  -159.990, Y  +567.494, Z    +0.000, E1   -35.052, E3 +391389.098}
SPL {X  -159.990, Y  +571.374, Z    +0.000, E1   -35.070, E3 +391400.801}
SPL {X  -159.990, Y  +575.771, Z    +0.000, E1   -35.064, E3 +391414.106}
SPL {X  -159.990, Y  +579.185, Z    +0.000, E1   -35.047, E3 +391424.454}
SPL {X  -159.990, Y  +581.944, Z    +0.000, E1   -35.051, E3 +391432.792}
SPL {X  -159.990, Y  +585.414, Z    +0.000, E1   -35.059, E3 +391443.275}
SPL {X  -159.990, Y  +590.166, Z    +0.000, E1   -35.084, E3 +391457.603}
SPL {X  -159.990, Y  +595.313, Z    +0.000, E1   -35.073, E3 +391473.182}
SPL {X  -159.990, Y  +600.543, Z    +0.000, E1   -35.091, E3 +391488.964}
SPL {X  -159.990, Y  +605.846, Z    +0.000, E1   -35.077, E3 +391505.015}
SPL {X  -159.990, Y  +609.372, Z    +0.000, E1   -35.047, E3 +391515.713}
SPL {X  -159.990, Y  +613.036, Z    +0.000, E1   -35.082, E3 +391526.748}
SPL {X  -159.990, Y  +617.577, Z    +0.000, E1   -35.061, E3 +391540.510}
SPL {X  -159.990, Y  +621.534, Z    +0.000, E1   -35.068, E3 +391552.444}
SPL {X  -159.990, Y  +625.237, Z    +0.000, E1   -35.062, E3 +391563.646}
SPL {X  -159.990, Y  +629.217, Z    +0.000, E1   -35.065, E3 +391575.703}
SPL {X  -159.990, Y  +632.566, Z    +0.000, E1   -35.044, E3 +391585.866}
SPL {X  -159.990, Y  +635.965, Z    +0.000, E1   -35.065, E3 +391596.109}
SPL {X  -159.990, Y  +640.633, Z    +0.000, E1   -35.080, E3 +391610.198}
SPL {X  -159.990, Y  +646.430, Z    +0.000, E1   -35.102, E3 +391627.699}
SPL {X  -159.990, Y  +651.502, Z    +0.000, E1   -35.058, E3 +391643.109}
SPL {X  -159.990, Y  +654.793, Z    +0.000, E1   -35.049, E3 +391653.072}
SPL {X  -159.990, Y  +657.535, Z    +0.000, E1   -35.049, E3 +391661.369}
SPL {X  -159.990, Y  +661.105, Z    +0.000, E1   -35.059, E3 +391672.149}
SPL {X  -159.990, Y  +665.311, Z    +0.000, E1   -35.064, E3 +391684.864}
SPL {X  -159.990, Y  +668.650, Z    +0.000, E1   -35.040, E3 +391695.003}
SPL {X  -159.990, Y  +671.288, Z    +0.000, E1   -35.046, E3 +391702.968}
SPL {X  -159.948, Y  +675.148, Z    +0.000, E1   -35.069, E3 +391714.603}
SPL {X  -159.752, Y  +680.228, Z    +0.000, E1   -35.050, E3 +391730.151}
SPL {X  -159.371, Y  +685.563, Z    +0.000, E1   -34.989, E3 +391746.662}
SPL {X  -158.886, Y  +690.264, Z    +0.000, E1   -34.888, E3 +391761.413}
SPL {X  -158.362, Y  +694.266, Z    +0.000, E1   -34.794, E3 +391774.087}
SPL {X  -157.614, Y  +698.973, Z    +0.000, E1   -34.690, E3 +391789.087}
SPL {X  -156.640, Y  +704.066, Z    +0.000, E1   -34.516, E3 +391805.513}
SPL {X  -155.835, Y  +707.723, Z    +0.000, E1   -34.344, E3 +391817.455}
SPL {X  -155.080, Y  +710.833, Z    +0.000, E1   -34.231, E3 +391827.605}
SPL {X  -153.949, Y  +715.047, Z    +0.000, E1   -29.578, E3 +391881.155}
ENDSPLINE

SPLINE
SPL {X  -158.529, Y  +693.075, Z    +0.000, E1   -15.996, E3 +391925.140}
SPL {X  -159.750, Y  +680.262, Z    +0.000, E1    -8.563, E3 +391933.551}
SPL {X  -159.973, Y  +673.798, Z    +0.000, E1    -4.600, E3 +391936.014}
SPL {X  -159.990, Y  +667.448, Z    +0.000, E1    -0.356, E3 +391937.794}
SPL {X  -159.990, Y  +662.686, Z    +0.000, E1    +3.472, E3 +391939.029}
SPL {X  -159.990, Y  +658.349, Z    +0.000, E1    +7.223, E3 +391940.397}
SPL {X  -159.990, Y  +653.910, Z    +0.000, E1   +11.344, E3 +391942.165}
SPL {X  -159.990, Y  +646.193, Z    +0.000, E1   +17.980, E3 +391946.634}
SPL {X  -159.990, Y  +621.124, Z    +0.000, E1   +32.598, E3 +391970.121}
SPL {X  -159.990, Y  +599.888, Z    +0.000, E1   +36.828, E3 +392007.360}
SPL {X  -159.990, Y  +595.346, Z    +0.000, E1   +36.880, E3 +392020.126}
SPL {X  -159.990, Y  +589.749, Z    +0.000, E1   +36.860, E3 +392035.999}
SPL {X  -159.990, Y  +585.754, Z    +0.000, E1   +36.838, E3 +392047.354}
SPL {X  -159.990, Y  +581.795, Z    +0.000, E1   +36.847, E3 +392058.567}
SPL {X  -159.990, Y  +576.165, Z    +0.000, E1   +36.887, E3 +392074.446}
SPL {X  -159.990, Y  +570.328, Z    +0.000, E1   +36.855, E3 +392091.019}
SPL {X  -159.990, Y  +566.126, Z    +0.000, E1   +36.841, E3 +392102.925}
SPL {X  -159.990, Y  +562.387, Z    +0.000, E1   +36.853, E3 +392113.458}
SPL {X  -159.990, Y  +557.944, Z    +0.000, E1   +36.859, E3 +392126.052}
SPL {X  -159.990, Y  +552.571, Z    +0.000, E1   +36.873, E3 +392141.256}
SPL {X  -159.990, Y  +548.223, Z    +0.000, E1   +36.832, E3 +392153.646}
SPL {X  -159.990, Y  +543.458, Z    +0.000, E1   +36.882, E3 +392167.049}
SPL {X  -159.990, Y  +537.639, Z    +0.000, E1   +36.860, E3 +392183.587}
SPL {X  -159.990, Y  +531.894, Z    +0.000, E1   +36.865, E3 +392199.876}
SPL {X  -159.990, Y  +525.940, Z    +0.000, E1   +36.859, E3 +392216.759}
SPL {X  -159.990, Y  +520.301, Z    +0.000, E1   +36.855, E3 +392232.735}
SPL {X  -159.990, Y  +516.005, Z    +0.000, E1   +36.824, E3 +392244.961}
SPL {X  -159.990, Y  +511.408, Z    +0.000, E1   +36.858, E3 +392257.930}
SPL {X  -159.990, Y  +505.756, Z    +0.000, E1   +36.857, E3 +392273.940}
SPL {X  -159.990, Y  +499.829, Z    +0.000, E1   +36.864, E3 +392290.745}
SPL {X  -159.990, Y  +498.054, Z    +0.000, E1   +35.692, E3 +392302.784}
ENDSPLINE

SPLINE
SPL {X  -159.990, Y  +506.994, Z    +0.000, E1   +30.162, E3 +392309.446}
ENDSPLINE

SPLINE
SPL {X  -159.990, Y  +502.084, Z    +0.000, E1   +31.057, E3 +392321.097}
SPL {X  -159.990, Y  +494.586, Z    +0.000, E1   +32.444, E3 +392337.700}
SPL {X  -159.990, Y  +487.723, Z    +0.000, E1   +33.658, E3 +392352.153}
SPL {X  -159.990, Y  +481.374, Z    +0.000, E1   +34.706, E3 +392365.357}
SPL {X  -159.990, Y  +475.503, Z    +0.000, E1   +35.597, E3 +392377.410}
SPL {X  -159.990, Y  +471.459, Z    +0.000, E1   +35.779, E3 +392388.256}
SPL {X  -159.990, Y  +466.474, Z    +0.000, E1   +35.796, E3 +392402.915}
SPL {X  -159.990, Y  +461.990, Z    +0.000, E1   +35.776, E3 +392416.150}
SPL {X  -159.990, Y  +457.385, Z    +0.000, E1   +35.788, E3 +392429.697}
SPL {X  -159.990, Y  +452.637, Z    +0.000, E1   +35.783, E3 +392443.689}
SPL {X  -159.990, Y  +446.982, Z    +0.000, E1   +35.815, E3 +392460.290}
SPL {X  -159.990, Y  +442.593, Z    +0.000, E1   +35.759, E3 +392473.299}
SPL {X  -159.990, Y  +439.109, Z    +0.000, E1   +35.781, E3 +392483.516}
SPL {X  -159.990, Y  +435.535, Z    +0.000, E1   +35.764, E3 +392494.067}
SPL {X  -159.990, Y  +431.100, Z    +0.000, E1   +35.807, E3 +392507.052}
SPL {X  -159.990, Y  +426.641, Z    +0.000, E1   +35.769, E3 +392520.239}
SPL {X  -159.990, Y  +422.627, Z    +0.000, E1   +35.788, E3 +392532.036}
SPL {X  -159.990, Y  +417.866, Z    +0.000, E1   +35.788, E3 +392546.050}
SPL {X  -159.990, Y  +413.498, Z    +0.000, E1   +35.779, E3 +392558.932}
SPL {X  -159.990, Y  +408.600, Z    +0.000, E1   +35.802, E3 +392573.319}
SPL {X  -159.990, Y  +403.496, Z    +0.000, E1   +35.787, E3 +392588.374}
SPL {X  -159.990, Y  +398.606, Z    +0.000, E1   +35.794, E3 +392602.762}
SPL {X  -159.990, Y  +394.138, Z    +0.000, E1   +35.778, E3 +392615.945}
SPL {X  -159.990, Y  +388.813, Z    +0.000, E1   +35.819, E3 +392631.557}
SPL {X  -159.990, Y  +383.172, Z    +0.000, E1   +35.789, E3 +392648.211}
SPL {X  -159.936, Y  +378.352, Z    +0.000, E1   +35.782, E3 +392662.450}
SPL {X  -159.790, Y  +374.497, Z    +0.000, E1   +35.735, E3 +392673.994}
SPL {X  -159.547, Y  +370.604, Z    +0.000, E1   +35.724, E3 +392685.679}
SPL {X  -159.134, Y  +365.969, Z    +0.000, E1   +35.644, E3 +392699.765}
SPL {X  -158.715, Y  +362.338, Z    +0.000, E1   +35.547, E3 +392710.973}
SPL {X  -158.237, Y  +358.884, Z    +0.000, E1   +35.480, E3 +392721.629}
SPL {X  -157.724, Y  +355.670, Z    +0.000, E1   +35.371, E3 +392731.664}
SPL {X  -157.185, Y  +352.671, Z    +0.000, E1   +35.292, E3 +392741.042}
SPL {X  -156.582, Y  +349.653, Z    +0.000, E1   +35.175, E3 +392750.576}
SPL {X  -155.743, Y  +345.880, Z    +0.000, E1   +35.068, E3 +392762.503}
SPL {X  -154.759, Y  +341.925, Z    +0.000, E1   +34.868, E3 +392775.209}
SPL {X  -154.305, Y  +340.232, Z    +0.000, E1   +28.975, E3 +392829.038}
ENDSPLINE

SPLINE
SPL {X  -158.456, Y  +360.399, Z    +0.000, E1   +16.490, E3 +392865.858}
SPL {X  -159.553, Y  +370.677, Z    +0.000, E1   +10.576, E3 +392873.618}
SPL {X  -159.960, Y  +379.402, Z    +0.000, E1    +5.303, E3 +392877.638}
SPL {X  -159.990, Y  +385.983, Z    +0.000, E1    +0.882, E3 +392879.711}
SPL {X  -159.990, Y  +390.933, Z    +0.000, E1    -2.877, E3 +392881.158}
SPL {X  -159.990, Y  +396.375, Z    +0.000, E1    -7.538, E3 +392882.933}
SPL {X  -159.990, Y  +405.219, Z    +0.000, E1   -15.296, E3 +392887.251}
SPL {X  -159.990, Y  +427.882, Z    +0.000, E1   -29.477, E3 +392908.930}
SPL {X  -159.990, Y  +452.779, Z    +0.000, E1   -35.077, E3 +392955.169}
SPL {X  -159.990, Y  +457.209, Z    +0.000, E1   -35.039, E3 +392968.629}
SPL {X  -159.990, Y  +460.708, Z    +0.000, E1   -35.045, E3 +392979.211}
SPL {X  -159.990, Y  +465.240, Z    +0.000, E1   -35.066, E3 +392992.887}
SPL {X  -159.990, Y  +470.278, Z    +0.000, E1   -35.063, E3 +393008.120}
SPL {X  -159.990, Y  +474.610, Z    +0.000, E1   -35.053, E3 +393021.219}
SPL {X  -159.990, Y  +479.424, Z    +0.000, E1   -35.081, E3 +393035.731}
SPL {X  -159.990, Y  +483.513, Z    +0.000, E1   -35.038, E3 +393048.185}
SPL {X  -159.990, Y  +487.181, Z    +0.000, E1   -35.054, E3 +393059.265}
SPL {X  -159.990, Y  +490.807, Z    +0.000, E1   -35.036, E3 +393070.267}
SPL {X  -159.990, Y  +493.669, Z    +0.000, E1   -35.034, E3 +393078.946}
SPL {X  -159.990, Y  +497.072, Z    +0.000, E1   -35.040, E3 +393089.233}
SPL {X  -159.990, Y  +500.395, Z    +0.000, E1   -35.033, E3 +393099.296}
SPL {X  -159.990, Y  +505.138, Z    +0.000, E1   -35.092, E3 +393113.533}
SPL {X  -159.990, Y  +510.443, Z    +0.000, E1   -35.051, E3 +393129.651}
SPL {X  -159.990, Y  +514.632, Z    +0.000, E1   -35.050, E3 +393142.321}
SPL {X  -159.990, Y  +518.055, Z    +0.000, E1   -35.037, E3 +393152.690}
SPL {X  -159.990, Y  +521.637, Z    +0.000, E1   -35.056, E3 +393163.500}
SPL {X  -159.990, Y  +526.246, Z    +0.000, E1   -35.065, E3 +393177.403}
SPL {X  -159.990, Y  +530.289, Z    +0.000, E1   -35.044, E3 +393189.690}
SPL {X  -159.990, Y  +534.797, Z    +0.000, E1   -35.069, E3 +393203.290}
SPL {X  -159.990, Y  +538.710, Z    +0.000, E1   -35.033, E3 +393215.187}
SPL {X  -159.990, Y  +542.114, Z    +0.000, E1   -35.053, E3 +393225.439}
SPL {X  -159.990, Y  +545.724, Z    +0.000, E1   -35.043, E3 +393236.364}
SPL {X  -159.990, Y  +549.546, Z    +0.000, E1   -35.061, E3 +393247.888}
SPL {X  -159.990, Y  +554.793, Z    +0.000, E1   -35.100, E3 +393263.651}
SPL {X  -159.990, Y  +560.931, Z    +0.000, E1   -35.098, E3 +393282.213}
SPL {X  -159.990, Y  +566.542, Z    +0.000, E1   -35.080, E3 +393299.220}
SPL {X  -159.990, Y  +571.374, Z    +0.000, E1   -35.070, E3 +393313.844}
SPL {X  -159.990, Y  +575.771, Z    +0.000, E1   -35.064, E3 +393327.149}
SPL {X  -159.990, Y  +580.750, Z    +0.000, E1   -35.087, E3 +393342.172}
SPL {X  -159.990, Y  +585.414, Z    +0.000, E1   -35.059, E3 +393356.318}
SPL {X  -159.990, Y  +588.716, Z    +0.000, E1   -35.047, E3 +393366.321}
SPL {X  -159.990, Y  +592.923, Z    +0.000, E1   -35.084, E3 +393378.985}
SPL {X  -159.990, Y  +598.554, Z    +0.000, E1   -35.088, E3 +393396.004}
SPL {X  -159.990, Y  +603.289, Z    +0.000, E1   -35.068, E3 +393410.332}
SPL {X  -159.990, Y  +606.793, Z    +0.000, E1   -35.050, E3 +393420.974}
SPL {X  -159.990, Y  +611.113, Z    +0.000, E1   -35.087, E3 +393433.965}
SPL {X  -159.990, Y  +616.690, Z    +0.000, E1   -35.089, E3 +393450.828}
SPL {X  -159.990, Y  +621.534, Z    +0.000, E1   -35.068, E3 +393465.487}
SPL {X  -159.990, Y  +626.426, Z    +0.000, E1   -35.093, E3 +393480.246}
SPL {X  -159.990, Y  +631.553, Z    +0.000, E1   -35.068, E3 +393495.805}
SPL {X  -159.990, Y  +636.917, Z    +0.000, E1   -35.095, E3 +393511.983}
SPL {X  -159.990, Y  +641.534, Z    +0.000, E1   -35.053, E3 +393526.011}
SPL {X  -159.990, Y  +646.430, Z    +0.000, E1   -35.102, E3 +393540.742}
SPL {X  -159.990, Y  +651.502, Z    +0.000, E1   -35.058, E3 +393556.152}
SPL {X  -159.990, Y  +654.793, Z    +0.000, E1   -35.049, E3 +393566.116}
SPL {X  -159.990, Y  +657.535, Z    +0.000, E1   -35.049, E3 +393574.412}
SPL {X  -159.990, Y  +661.105, Z    +0.000, E1   -35.059, E3 +393585.192}
SPL {X  -159.990, Y  +665.311, Z    +0.000, E1   -35.064, E3 +393597.907}
SPL {X  -159.990, Y  +670.193, Z    +0.000, E1   -35.076, E3 +393612.654}
SPL {X  -159.948, Y  +675.148, Z    +0.000, E1   -35.069, E3 +393627.646}
SPL {X  -159.805, Y  +679.202, Z    +0.000, E1   -35.029, E3 +393640.079}
SPL {X  -159.584, Y  +682.885, Z    +0.000, E1   -34.997, E3 +393651.439}
SPL {X  -159.292, Y  +686.426, Z    +0.000, E1   -34.947, E3 +393662.440}
SPL {X  -158.886, Y  +690.264, Z    +0.000, E1   -34.888, E3 +393674.457}
SPL {X  -158.362, Y  +694.266, Z    +0.000, E1   -34.794, E3 +393687.130}
SPL {X  -157.614, Y  +698.973, Z    +0.000, E1   -34.690, E3 +393702.131}
SPL {X  -156.640, Y  +704.066, Z    +0.000, E1   -34.516, E3 +393718.556}
SPL {X  -155.835, Y  +707.723, Z    +0.000, E1   -34.344, E3 +393730.498}
SPL {X  -155.080, Y  +710.833, Z    +0.000, E1   -34.231, E3 +393740.648}
SPL {X  -153.949, Y  +715.047, Z    +0.000, E1   -29.578, E3 +393794.198}
ENDSPLINE

SPLINE
SPL {X  -158.529, Y  +693.075, Z    +0.000, E1   -15.996, E3 +393838.183}
SPL {X  -159.750, Y  +680.262, Z    +0.000, E1    -8.563, E3 +393846.594}
SPL {X  -159.973, Y  +673.798, Z    +0.000, E1    -4.600, E3 +393849.058}
SPL {X  -159.990, Y  +668.863, Z    +0.000, E1    -1.298, E3 +393850.497}
SPL {X  -159.990, Y  +663.839, Z    +0.000, E1    +2.454, E3 +393851.758}
SPL {X  -159.990, Y  +658.349, Z    +0.000, E1    +7.223, E3 +393853.440}
SPL {X  -159.990, Y  +653.910, Z    +0.000, E1   +11.344, E3 +393855.208}
SPL {X  -159.990, Y  +646.193, Z    +0.000, E1   +17.980, E3 +393859.677}
SPL {X  -159.990, Y  +621.124, Z    +0.000, E1   +32.598, E3 +393883.164}
SPL {X  -159.990, Y  +597.855, Z    +0.000, E1   +36.862, E3 +393926.084}
SPL {X  -159.990, Y  +593.971, Z    +0.000, E1   +36.841, E3 +393937.116}
SPL {X  -159.990, Y  +589.749, Z    +0.000, E1   +36.860, E3 +393949.043}
SPL {X  -159.990, Y  +585.754, Z    +0.000, E1   +36.838, E3 +393960.398}
SPL {X  -159.990, Y  +581.795, Z    +0.000, E1   +36.847, E3 +393971.610}
SPL {X  -159.990, Y  +577.286, Z    +0.000, E1   +36.853, E3 +393984.367}
SPL {X  -159.990, Y  +572.409, Z    +0.000, E1   +36.854, E3 +393998.179}
SPL {X  -159.990, Y  +567.110, Z    +0.000, E1   +36.868, E3 +394013.140}
SPL {X  -159.990, Y  +562.387, Z    +0.000, E1   +36.853, E3 +394026.502}
SPL {X  -159.990, Y  +557.944, Z    +0.000, E1   +36.859, E3 +394039.095}
SPL {X  -159.990, Y  +553.661, Z    +0.000, E1   +36.844, E3 +394051.259}
SPL {X  -159.990, Y  +549.195, Z    +0.000, E1   +36.856, E3 +394063.894}
SPL {X  -159.990, Y  +544.733, Z    +0.000, E1   +36.845, E3 +394076.540}
SPL {X  -159.990, Y  +539.889, Z    +0.000, E1   +36.872, E3 +394090.225}
SPL {X  -159.990, Y  +534.469, Z    +0.000, E1   +36.855, E3 +394105.622}
SPL {X  -159.990, Y  +530.428, Z    +0.000, E1   +36.821, E3 +394117.156}
SPL {X  -159.990, Y  +525.940, Z    +0.000, E1   +36.859, E3 +394129.802}
SPL {X  -159.990, Y  +520.301, Z    +0.000, E1   +36.855, E3 +394145.778}
SPL {X  -159.990, Y  +516.005, Z    +0.000, E1   +36.824, E3 +394158.005}
SPL {X  -159.990, Y  +511.408, Z    +0.000, E1   +36.858, E3 +394170.974}
SPL {X  -159.990, Y  +505.756, Z    +0.000, E1   +36.857, E3 +394186.983}
SPL {X  -159.990, Y  +499.829, Z    +0.000, E1   +36.864, E3 +394203.788}
SPL {X  -159.990, Y  +498.054, Z    +0.000, E1   +35.692, E3 +394215.827}
ENDSPLINE

SPLINE
SPL {X  -159.990, Y  +505.140, Z    +0.000, E1   +30.523, E3 +394226.854}
ENDSPLINE

SPLINE
SPL {X  -159.990, Y  +497.800, Z    +0.000, E1   +31.845, E3 +394243.810}
SPL {X  -159.990, Y  +492.180, Z    +0.000, E1   +32.851, E3 +394255.946}
SPL {X  -159.990, Y  +486.073, Z    +0.000, E1   +33.960, E3 +394268.582}
SPL {X  -159.990, Y  +477.314, Z    +0.000, E1   +35.342, E3 +394286.760}
SPL {X  -159.990, Y  +471.459, Z    +0.000, E1   +35.779, E3 +394301.299}
SPL {X  -159.990, Y  +467.485, Z    +0.000, E1   +35.768, E3 +394313.029}
SPL {X  -159.990, Y  +462.739, Z    +0.000, E1   +35.799, E3 +394326.957}
SPL {X  -159.990, Y  +457.385, Z    +0.000, E1   +35.788, E3 +394342.740}
SPL {X  -159.990, Y  +452.637, Z    +0.000, E1   +35.783, E3 +394356.732}
SPL {X  -159.990, Y  +448.227, Z    +0.000, E1   +35.776, E3 +394369.729}
SPL {X  -159.990, Y  +443.707, Z    +0.000, E1   +35.784, E3 +394383.024}
SPL {X  -159.990, Y  +439.109, Z    +0.000, E1   +35.781, E3 +394396.560}
SPL {X  -159.990, Y  +434.400, Z    +0.000, E1   +35.789, E3 +394410.415}
SPL {X  -159.990, Y  +430.115, Z    +0.000, E1   +35.777, E3 +394423.032}
SPL {X  -159.990, Y  +425.407, Z    +0.000, E1   +35.800, E3 +394436.871}
SPL {X  -159.990, Y  +420.199, Z    +0.000, E1   +35.790, E3 +394452.225}
SPL {X  -159.990, Y  +414.514, Z    +0.000, E1   +35.815, E3 +394468.924}
SPL {X  -159.990, Y  +408.600, Z    +0.000, E1   +35.802, E3 +394486.363}
SPL {X  -159.990, Y  +403.496, Z    +0.000, E1   +35.787, E3 +394501.418}
SPL {X  -159.990, Y  +398.606, Z    +0.000, E1   +35.794, E3 +394515.805}
SPL {X  -159.990, Y  +394.138, Z    +0.000, E1   +35.778, E3 +394528.988}
SPL {X  -159.990, Y  +390.065, Z    +0.000, E1   +35.780, E3 +394540.978}
SPL {X  -159.990, Y  +385.506, Z    +0.000, E1   +35.789, E3 +394554.384}
SPL {X  -159.976, Y  +380.359, Z    +0.000, E1   +35.797, E3 +394569.533}
SPL {X  -159.831, Y  +375.358, Z    +0.000, E1   +35.763, E3 +394584.423}
SPL {X  -159.547, Y  +370.604, Z    +0.000, E1   +35.724, E3 +394598.723}
SPL {X  -159.134, Y  +365.969, Z    +0.000, E1   +35.644, E3 +394612.808}
SPL {X  -158.715, Y  +362.338, Z    +0.000, E1   +35.547, E3 +394624.016}
SPL {X  -158.237, Y  +358.884, Z    +0.000, E1   +35.480, E3 +394634.673}
SPL {X  -157.724, Y  +355.670, Z    +0.000, E1   +35.371, E3 +394644.707}
SPL {X  -157.185, Y  +352.671, Z    +0.000, E1   +35.292, E3 +394654.086}
SPL {X  -156.582, Y  +349.653, Z    +0.000, E1   +35.175, E3 +394663.619}
SPL {X  -155.743, Y  +345.880, Z    +0.000, E1   +35.068, E3 +394675.546}
SPL {X  -154.759, Y  +341.925, Z    +0.000, E1   +34.868, E3 +394688.252}
SPL {X  -154.305, Y  +340.232, Z    +0.000, E1   +28.975, E3 +394742.082}
ENDSPLINE

